// SIMATIC STEP 7 (V5.x) project S7_Mafra
// CPU: CPU 312
// CPU: CPU 312
// station: P_ADR_BUS
// station: Hardware
// station: Mafra_Praha
// station: P_ADR_BUS
// station: Hardware
// station: Mafra_Olomouc
// station: P_ADR_BUS
// station: Configuration
// station: P_ADR_BUS
// station: Configuration
// program: S7 Program(2)
// program: S7 Program(2)

SYMBOL_TABLE
"Události"	DB 100	DB 100
"DB_Chyby"	DB 101	DB 101
"DB_Ruèni povely pro HMI"	DB 120	DB 120
"DB_Data Hmi"	DB 140	DB 140
"Globální øízení"	FC 10	FC 10
"Váleèkové dopravníky"	FC 20	FC 20
"Data HMI"	FC 30	FC 30
"Chyby"	FC 40	FC 40
"Komunikace"	FC 50	FC 50
"Pohony P1,P2.1 a P2.2 OK"	I 0.0	BOOL	// Pohony dopr.P1 , toèny P2.2 a dopravníku P2.2 jsou OK
"Pohony P3,P4.1 a P4.2 OK"	I 0.1	BOOL	// Pohony dopr.P3 , toèny P4.1 a dopravníku P4.2 jsou OK
"Pohony P7,P8,P9 OK"	I 0.2	BOOL	// Pohony dopr.P7,P8,P9 jsou OK
"Silovka OK"	I 0.3	BOOL	// Silové obvody zapnuty
"Reset"	I 0.4	BOOL	// Reset programu
"Vynut NOT-Aus rozvadìè"	I 0.5	BOOL	// Vypnutý hlavní NOT-AUS na rozvadìèi
"NOT-AUS 1"	I 0.6	BOOL	// Vypnut NOT-AUS 1
"NOT-AUS 2"	I 0.7	BOOL	// Vypnut NOT-AUS 2
"Balík na konci P1"	I 1.0	BOOL	// Balík dojet na konci dopravníku 1
"Balík na konci P2.2"	I 1.1	BOOL	// Balík dojet na konci dopravníku 2.2
"Toèna 2.1 nájezd"	I 1.2	BOOL	// Toèna P2.1 pozice nájezd
"Toèna 2.1 výjezd"	I 1.3	BOOL	// Toèna P2.1 pozice výjezd
"Balík na konci P3"	I 1.4	BOOL	// Balík dojet na konci dopravníku 3
"Balík na konci P4.2"	I 1.5	BOOL	// Balík dojet na konci dopravníku 4.2
"Toèna 4.1 nájezd"	I 1.6	BOOL	// Toèna P4.1 pozice nájezd
"Toèna 4.1 výjezd"	I 1.7	BOOL	// Toèna P4.1 pozice výjezd
"Balík na konci P5"	I 2.0	BOOL	// Balík dojet na konci dopravníku 5
"Balík na konci P6"	I 2.1	BOOL	// Balík dojet na konci dopravníku 6
"Balík na konci P7"	I 2.2	BOOL	// Balík dojet na konci dopravníku 7
"Balík na konci P8"	I 2.3	BOOL	// Balík dojet na konci dopravníku 8
"S024"	I 2.4	BOOL	// stop na D2
"rezerva 1"	I 2.5	BOOL
"rezerva 2"	I 2.6	BOOL
"rezerva 3"	I 2.7	BOOL
"Komunikace vstup 1"	I 3.0	BOOL
"Komunikace vstup2"	I 3.1	BOOL
"Komunikace vstup 3"	I 3.2	BOOL
"Komunikace vstup 4"	I 3.3	BOOL
"rezerva 4"	I 3.4	BOOL
"rezerva 5"	I 3.5	BOOL
"rezerva 6"	I 3.6	BOOL
"rezerva 7"	I 3.7	BOOL
"True"	M 0.3	BOOL
"Automat"	M 1.0	BOOL	// Automatický chod stroje
"Chyba"	M 2.0	BOOL	// vyhlašení chybového stavu stroje
"PM21"	M 2.1	BOOL	// pomocný merkr
"Houkat"	M 4.4	BOOL	// pomocný merkr pro houkaèku
"Toèna P2 Stop nájezd"	M 6.0	BOOL
"Toèna P2 Stop výjezd"	M 6.1	BOOL
"Toèna P4 Stop nájezd"	M 6.2	BOOL
"Toèna P4 Stop výjezd"	M 6.4	BOOL
"M-Toèna 2 nájezd"	M 7.0	BOOL
"M-Toèna 2 výjezd"	M 7.1	BOOL
"M-Toèna 4 výjezd"	M 7.2	BOOL
"M-Toèna 4 nájezd"	M 7.3	BOOL
"Pøesun Balièka-P1"	M 20.0	BOOL	// pomocny merk pøesunu balíku z balièky na toènu
"Pøesun z Toèny na P3"	M 20.1	BOOL	// set a reset pøesunu balíku z toèny na dopravník P3
"Pøesun P3 - Toèna P4."	M 20.2	BOOL	// set a reset pøesunu z dopravníku P3 na toènu P4.1
"Pøesun Toèna P4.1-P5"	M 20.3	BOOL	// set a reset pøesunu z Toèny P4.1 na dopravník P5
"Pøesun P5-P6"	M 20.4	BOOL	// set a reset pøesunu balíku z P5 na P6
"Pøesun P6-P7"	M 20.5	BOOL	// set a reset pøesunu z dopravníku P6 na P7
"Pøesun P7-P8"	M 20.6	BOOL	// set a reset pøesunu z dopravníku P7 na P8
"CYC_INT5"	OB 35	OB 35	// Cyclic Interrupt 5
"I/O_FLT1"	OB 82	OB 82	// I/O Point Fault 1
"OBNL_FLT"	OB 85	OB 85	// OB Not Loaded Fault
"RACK_FLT"	OB 86	OB 86	// Loss of Rack Fault
"Complete Restart"	OB 100	OB 100
"Programming Error"	OB 121	OB 121
"Module Access Error"	OB 122	OB 122
"Dopravník 1 vpøed"	Q 4.0	BOOL	// Start dopravníku 1
"Toèna P2.1 nájezd"	Q 4.1	BOOL	// Toèna P2.1 nájezd
"Toèna P2.1 výjezd"	Q 4.2	BOOL	// Toèna P2.1 výjezd
"Toèna P2.1 brzda"	Q 4.3	BOOL	// Toèna P2.1 bzrda
"Dopravník 2.2 vpøed"	Q 4.4	BOOL	// Start dopravníku 2.2
"Dopravník 3 vpøed"	Q 4.5	BOOL	// Start dopravníku 3
"Toèna P4.1 nájezd"	Q 4.6	BOOL	// Toèna P4.1 nájezd
"Toèna P4.1 výjezd"	Q 4.7	BOOL	// Toèna P4.1 výjezd
"Toèna P4.1 brzda"	Q 5.0	BOOL	// Toèna P4.1 bzrda
"Dopravník P4.2 vpøed"	Q 5.1	BOOL	// Start dopravníku 4.2
"Dopravník 5 vpøed"	Q 5.2	BOOL	// Start dopravníku 5
"Dopravník 6 vpøed"	Q 5.3	BOOL	// Start dopravníku 6
"Dopravník 7 vpøed"	Q 5.4	BOOL	// Start dopravníku 7
"Dopravník 8 vpøed"	Q 5.5	BOOL	// Start dopravníku 8
"rezerva 8"	Q 5.6	BOOL
"rezerva 9"	Q 5.7	BOOL
"Signálka Zapnuto"	Q 6.0	BOOL	// Signálk zapnuto
"rezerva 10"	Q 6.1	BOOL
"rezerva 11"	Q 6.2	BOOL
"rezerva 12"	Q 6.3	BOOL
"Maják zelená"	Q 6.4	BOOL	// Signalizaèní sloupek - zelená
"Maják oranžová"	Q 6.5	BOOL	// Signalizaèní sloupek - oranžová
"Maják èervená"	Q 6.6	BOOL	// Signalizaèní sloupek - èervená
"Houkaèka"	Q 6.7	BOOL	// Signalizaèní sloupek - houkaèka
"Komunikace výstup 1"	Q 7.0	BOOL
"Komunikace výstup 2"	Q 7.1	BOOL
"Komunikace výstup 3"	Q 7.2	BOOL
"Komunikace-Plná linka"	Q 7.3	BOOL
"rezerva 13"	Q 7.4	BOOL
"rezerva 14"	Q 7.5	BOOL
"rezerva 15"	Q 7.6	BOOL
"rezerva 16"	Q 7.7	BOOL
"T-Automat"	T 0	TIMER	// zpoždìné spuštìní automatu
"T-Balík na konci P8"	T 2	TIMER	// Zpoždìný start pøesunu
"T-Pozor"	T 3	TIMER	// upozornìní na spouštìjící se automat
"T-S011"	T 10	TIMER	// balik dojet na konci D2
"T-S015"	T 11	TIMER
"T-Balík na konci"	T 12	TIMER
"T-Možno otoèit toènu"	T 13	TIMER
"T-Možno otoèit toènu P4"	T 14	TIMER
"T-S010"	T 15	TIMER	// balík dojet na konci skluzu
"T-Pøesun Balièka-P2.2"	T 20	TIMER	// èasovaè pro vyhlášení pøíliš dlouhého pøesunu
"T-Pøesun P2.2-P3"	T 21	TIMER	// èasovaè pro vyhlášení pøíliš dlouhého pøesunu
"T-Pøesun P3-P4.2"	T 22	TIMER	// èasovaè pro vyhlášení pøíliš dlouhého pøesunu
"T-Pøesun P4.2-P5"	T 23	TIMER	// èasovaè pro vyhlášení pøíliš dlouhého pøesunu
"T-Pøesun P5-P6"	T 24	TIMER	// èasovaè pro vyhlášení pøíliš dlouhého pøesunu
"T-Pøesun P6-P7"	T 25	TIMER	// èasovaè pro vyhlášení pøíliš dlouhého pøesunu
"T-Pøesun P7-P8"	T 26	TIMER	// èasovaè pro vyhlášení pøíliš dlouhého pøesunu
"T-Otaèení Toèny P2.1"	T 27	TIMER	// èasovaè pro vyhlášení pøíliš dlouhého otáèení toèny
"T-Otáèení toèny P4.1"	T 28	TIMER	// èasovaè pro vyhlášení pøíliš dlouhého otáèení toèny
"T-S014"	T 30	TIMER	// balik dojet na konci dopravniku
"T--S015"	T 31	TIMER	// balík na konci D4
"T-S020"	T 32	TIMER	// balík na konci D5
"T-S021"	T 33	TIMER	// balík na konci D6
"T-S022"	T 34	TIMER	// balík na konci D7
"T--S011"	T 35	TIMER
"T-S024"	T 37	TIMER	// Stop na D2
"VAT_1"	VAT 1	
END_SYMBOL_TABLE

FUNCTION "Globální øízení" : VOID	// FC 10
VERSION : 0.1
BEGIN
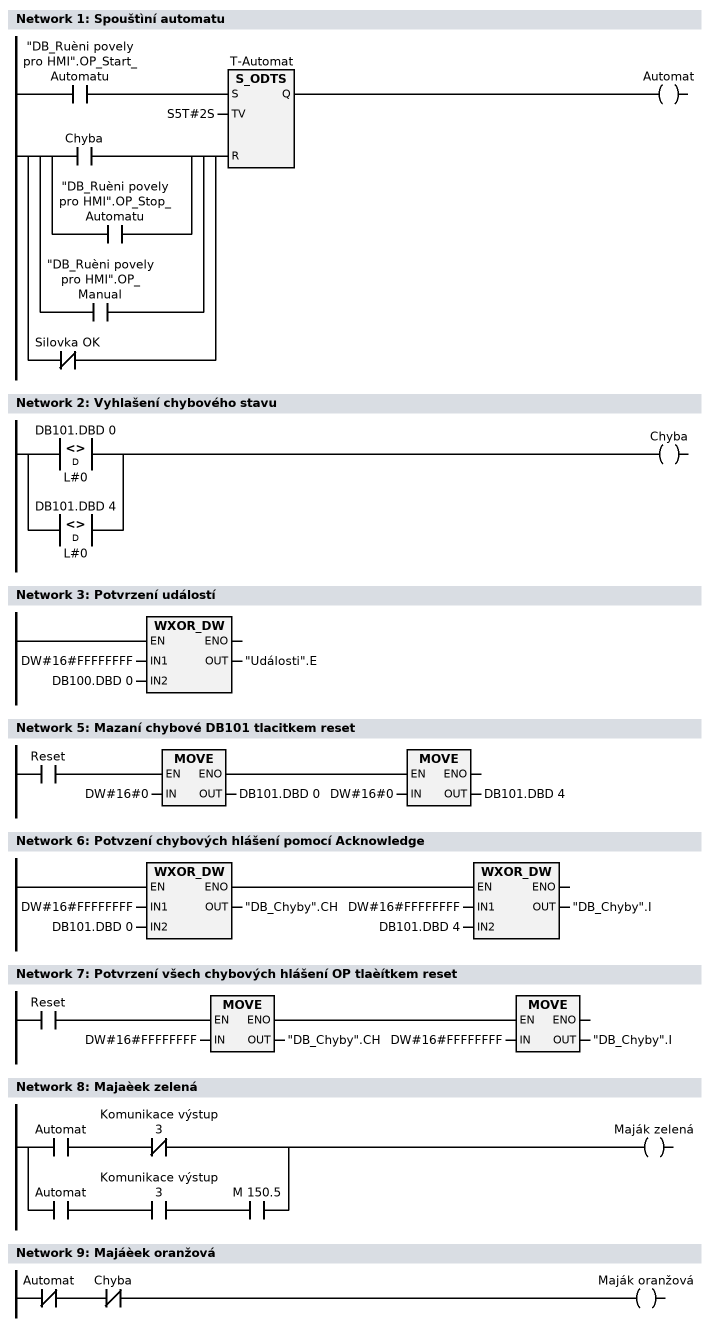
NETWORK
TITLE = Spouštìní automatu 
      A     "DB_Ruèni povely pro HMI".OP_Start_Automatu;
      L     S5T#2S;
      SS    "T-Automat";
      A(;
      O     "Chyba";
      O     "DB_Ruèni povely pro HMI".OP_Stop_Automatu;
      O     "DB_Ruèni povely pro HMI".OP_Manual;
      ON    "Silovka OK";
      );
      R     "T-Automat";
      NOP   0;
      NOP   0;
      A     "T-Automat";
      =     "Automat";
NETWORK
TITLE = Vyhlašení chybového stavu 
      O(;
      L     DB101.DBD 0;
      L     L#0;
      <>D;
      );
      O(;
      L     DB101.DBD 4;
      L     L#0;
      <>D;
      );
      =     "Chyba";
NETWORK
TITLE = Potvrzení událostí
      L     DW#16#FFFFFFFF;
      L     DB100.DBD 0;
      XOD;
      T     "Události".E;
      NOP   0;
NETWORK
TITLE = Akustická signalizace 
      A(;
      O(;
      A     "Chyba";
      FP    "PM21";
      S     "Houkat";
      A     "Reset";
      R     "Houkat";
      A     "Houkat";
      );
      O(;
      A     "DB_Ruèni povely pro HMI".OP_Start_Automatu;
      L     S5T#2S;
      SE    "T-Pozor";
      A(;
      O     "Chyba";
      O     "DB_Ruèni povely pro HMI".OP_Manual;
      O     "DB_Ruèni povely pro HMI".OP_Stop_Automatu;
      O     "Automat";
      );
      R     "T-Pozor";
      NOP   0;
      NOP   0;
      A     "T-Pozor";
      );
      );
      A     M 150.5;
      =     "Houkaèka";
NETWORK
TITLE = Mazaní chybové DB101 tlacitkem reset
      A(;
      A     "Reset";
      JNB   _001;
      L     DW#16#0;
      T     DB101.DBD 0;
      SET;
      SAVE;
      CLR;
_001: A     BR;
      );
      JNB   _002;
      L     DW#16#0;
      T     DB101.DBD 4;
_002: NOP   0;
NETWORK
TITLE = Potvzení chybových hlášení pomocí Acknowledge
      A(;
      L     DW#16#FFFFFFFF;
      L     DB101.DBD 0;
      XOD;
      T     "DB_Chyby".CH;
      SET;
      SAVE;
      CLR;
      A     BR;
      );
      JNB   _003;
      L     DW#16#FFFFFFFF;
      L     DB101.DBD 4;
      XOD;
      T     "DB_Chyby".I;
_003: NOP   0;
NETWORK
TITLE = Potvrzení všech chybových hlášení OP tlaèítkem reset
      A(;
      A     "Reset";
      JNB   _004;
      L     DW#16#FFFFFFFF;
      T     "DB_Chyby".CH;
      SET;
      SAVE;
      CLR;
_004: A     BR;
      );
      JNB   _005;
      L     DW#16#FFFFFFFF;
      T     "DB_Chyby".I;
_005: NOP   0;
NETWORK
TITLE = Majaèek zelená 
      A     "Automat";
      AN    "Komunikace výstup 3";
      O;
      A     "Automat";
      A     "Komunikace výstup 3";
      A     M 150.5;
      =     "Maják zelená";
NETWORK
TITLE = Majáèek oranžová 
      AN    "Automat";
      AN    "Chyba";
      =     "Maják oranžová";
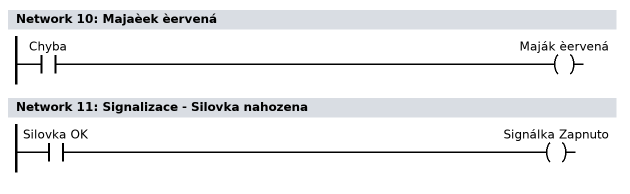
NETWORK
TITLE = Majaèek èervená 
      A     "Chyba";
      =     "Maják èervená";
NETWORK
TITLE = Signalizace - Silovka nahozena
      A     "Silovka OK";
      =     "Signálka Zapnuto";
END_FUNCTION

FUNCTION "Váleèkové dopravníky" : VOID	// FC 20
VERSION : 0.1
BEGIN
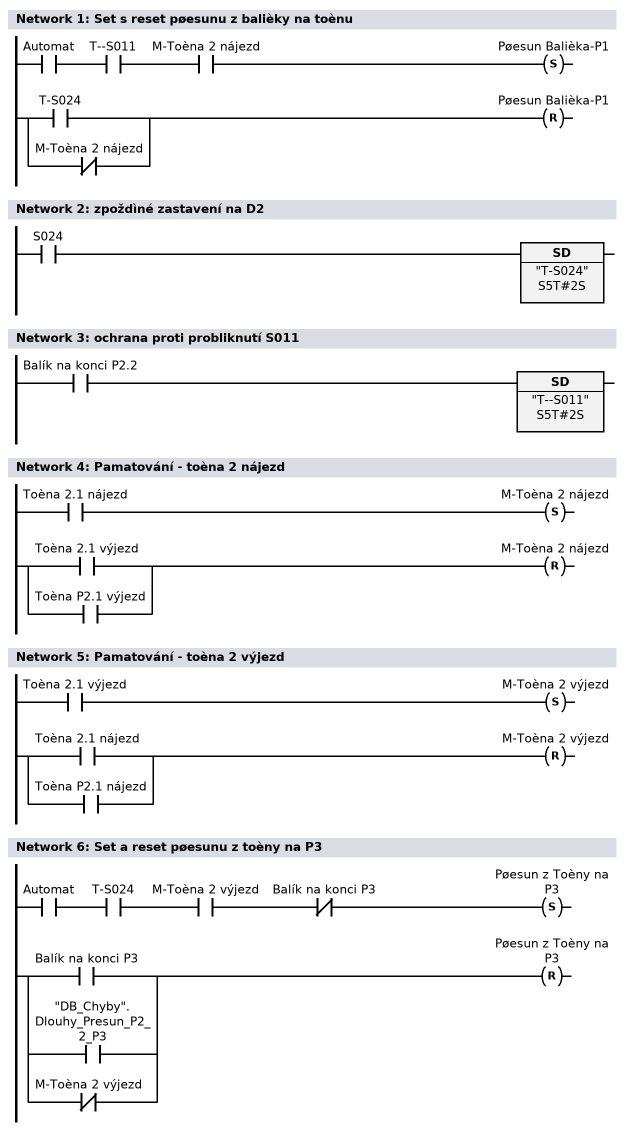
NETWORK
TITLE = Set s reset pøesunu z balièky na toènu
      A     "Automat";
      A     "T--S011";
      A     "M-Toèna 2 nájezd";
      S     "Pøesun Balièka-P1";
      A(;
      O     "T-S024";
      ON    "M-Toèna 2 nájezd";
      );
      R     "Pøesun Balièka-P1";
      NOP   0;
NETWORK
TITLE = zpoždìné zastavení na D2
      A     "S024";
      L     S5T#2S;
      SD    "T-S024";
NETWORK
TITLE = ochrana proti probliknutí S011
      A     "Balík na konci P2.2";
      L     S5T#2S;
      SD    "T--S011";
NETWORK
TITLE = Pamatování - toèna 2 nájezd
      A     "Toèna 2.1 nájezd";
      S     "M-Toèna 2 nájezd";
      A(;
      O     "Toèna 2.1 výjezd";
      O     "Toèna P2.1 výjezd";
      );
      R     "M-Toèna 2 nájezd";
      NOP   0;
NETWORK
TITLE = Pamatování - toèna 2 výjezd
      A     "Toèna 2.1 výjezd";
      S     "M-Toèna 2 výjezd";
      A(;
      O     "Toèna 2.1 nájezd";
      O     "Toèna P2.1 nájezd";
      );
      R     "M-Toèna 2 výjezd";
      NOP   0;
NETWORK
TITLE = Set a reset pøesunu z toèny na P3
      A     "Automat";
      A     "T-S024";
      A     "M-Toèna 2 výjezd";
      AN    "Balík na konci P3";
      S     "Pøesun z Toèny na P3";
      A(;
      O     "Balík na konci P3";
      O     "DB_Chyby".Dlouhy_Presun_P2_2_P3;
      ON    "M-Toèna 2 výjezd";
      );
      R     "Pøesun z Toèny na P3";
      NOP   0;
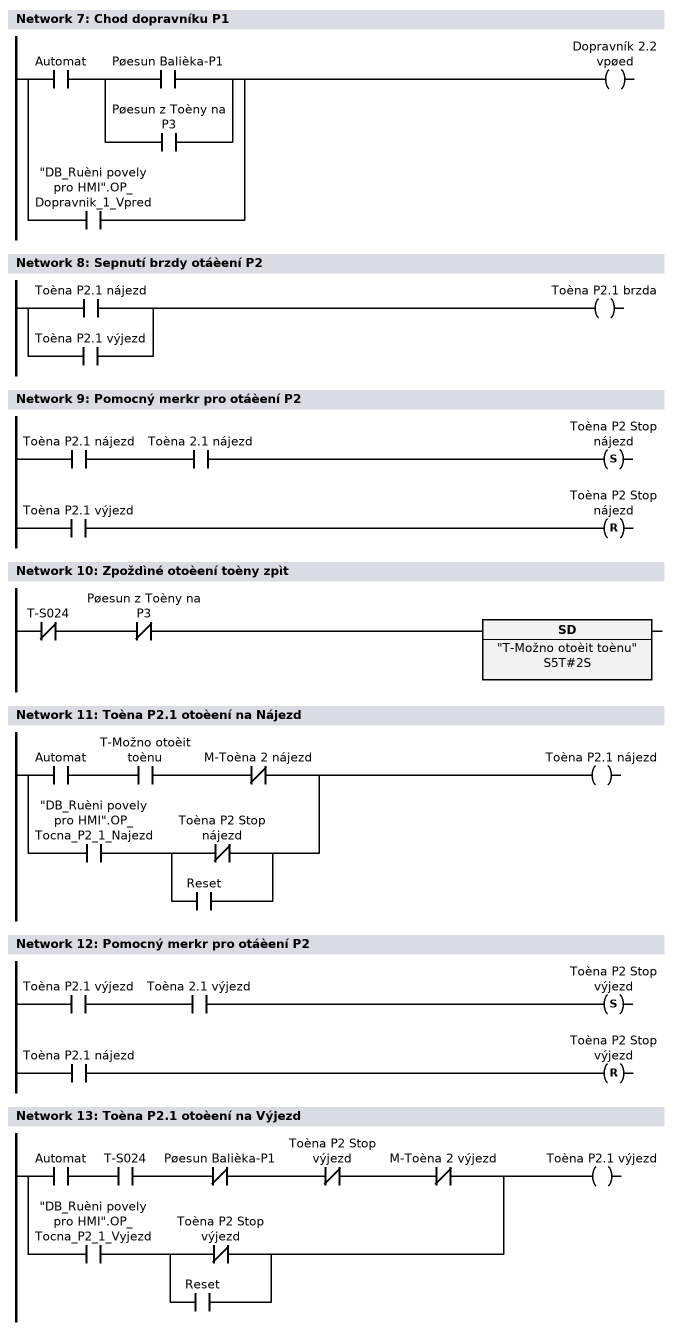
NETWORK
TITLE = Chod dopravníku P1
      A     "Automat";
      A(;
      O     "Pøesun Balièka-P1";
      O     "Pøesun z Toèny na P3";
      );
      O     "DB_Ruèni povely pro HMI".OP_Dopravnik_1_Vpred;
      =     "Dopravník 2.2 vpøed";
NETWORK
TITLE = Sepnutí brzdy otáèení P2
      O     "Toèna P2.1 nájezd";
      O     "Toèna P2.1 výjezd";
      =     "Toèna P2.1 brzda";
NETWORK
TITLE = Pomocný merkr pro otáèení P2
//Kvùli prokmitu toèny 
      A     "Toèna P2.1 nájezd";
      A     "Toèna 2.1 nájezd";
      S     "Toèna P2 Stop nájezd";
      A     "Toèna P2.1 výjezd";
      R     "Toèna P2 Stop nájezd";
      NOP   0;
NETWORK
TITLE = Zpoždìné otoèení toèny zpìt
      AN    "T-S024";
      AN    "Pøesun z Toèny na P3";
      L     S5T#2S;
      SD    "T-Možno otoèit toènu";
NETWORK
TITLE = Toèna P2.1 otoèení na Nájezd
      A     "Automat";
      A     "T-Možno otoèit toènu";
      AN    "M-Toèna 2 nájezd";
      O;
      A     "DB_Ruèni povely pro HMI".OP_Tocna_P2_1_Najezd;
      A(;
      ON    "Toèna P2 Stop nájezd";
      O     "Reset";
      );
      =     "Toèna P2.1 nájezd";
NETWORK
TITLE = Pomocný merkr pro otáèení P2
//Kvùli prokmitu toèny 
      A     "Toèna P2.1 výjezd";
      A     "Toèna 2.1 výjezd";
      S     "Toèna P2 Stop výjezd";
      A     "Toèna P2.1 nájezd";
      R     "Toèna P2 Stop výjezd";
      NOP   0;
NETWORK
TITLE = Toèna P2.1 otoèení na Výjezd
      A     "Automat";
      A     "T-S024";
      AN    "Pøesun Balièka-P1";
      AN    "Toèna P2 Stop výjezd";
      AN    "M-Toèna 2 výjezd";
      O;
      A     "DB_Ruèni povely pro HMI".OP_Tocna_P2_1_Vyjezd;
      A(;
      ON    "Toèna P2 Stop výjezd";
      O     "Reset";
      );
      =     "Toèna P2.1 výjezd";
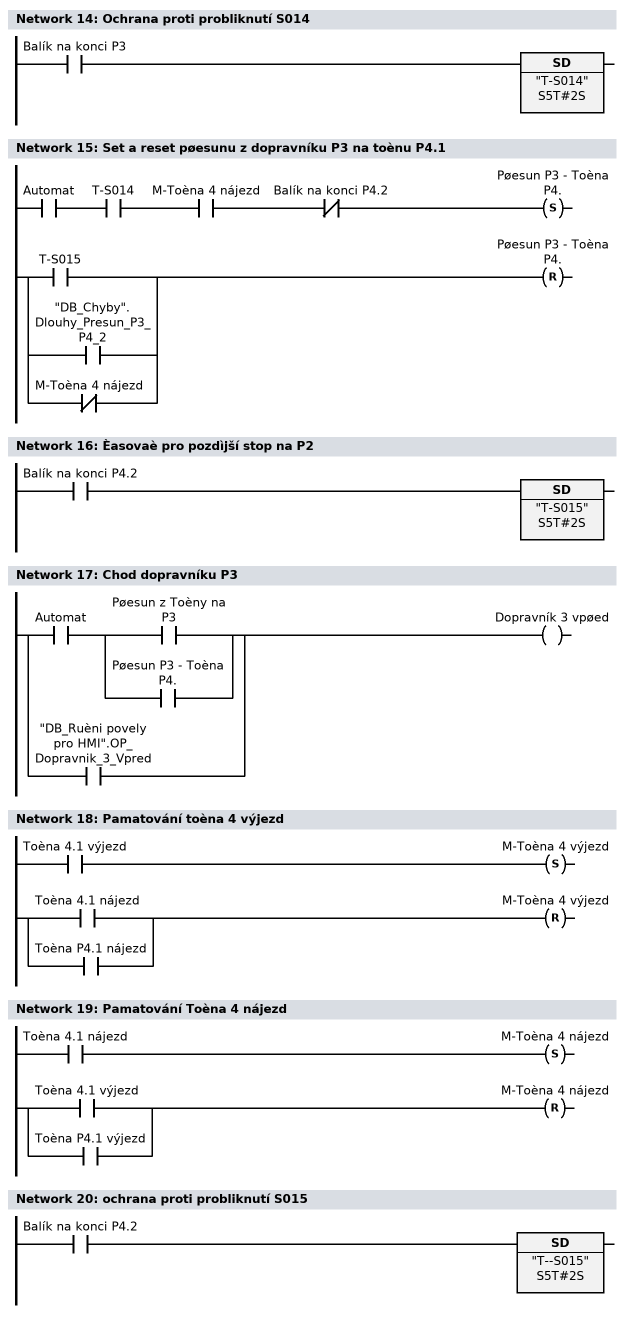
NETWORK
TITLE = Ochrana proti probliknutí S014
      A     "Balík na konci P3";
      L     S5T#2S;
      SD    "T-S014";
NETWORK
TITLE = Set a reset pøesunu z dopravníku P3 na toènu P4.1
      A     "Automat";
      A     "T-S014";
      A     "M-Toèna 4 nájezd";
      AN    "Balík na konci P4.2";
      S     "Pøesun P3 - Toèna P4.";
      A(;
      O     "T-S015";
      O     "DB_Chyby".Dlouhy_Presun_P3_P4_2;
      ON    "M-Toèna 4 nájezd";
      );
      R     "Pøesun P3 - Toèna P4.";
      NOP   0;
NETWORK
TITLE = Èasovaè pro pozdìjší stop na P2
      A     "Balík na konci P4.2";
      L     S5T#2S;
      SD    "T-S015";
NETWORK
TITLE = Chod dopravníku P3
      A     "Automat";
      A(;
      O     "Pøesun z Toèny na P3";
      O     "Pøesun P3 - Toèna P4.";
      );
      O     "DB_Ruèni povely pro HMI".OP_Dopravnik_3_Vpred;
      =     "Dopravník 3 vpøed";
NETWORK
TITLE = Pamatování toèna 4 výjezd
      A     "Toèna 4.1 výjezd";
      S     "M-Toèna 4 výjezd";
      A(;
      O     "Toèna 4.1 nájezd";
      O     "Toèna P4.1 nájezd";
      );
      R     "M-Toèna 4 výjezd";
      NOP   0;
NETWORK
TITLE = Pamatování Toèna 4 nájezd
      A     "Toèna 4.1 nájezd";
      S     "M-Toèna 4 nájezd";
      A(;
      O     "Toèna 4.1 výjezd";
      O     "Toèna P4.1 výjezd";
      );
      R     "M-Toèna 4 nájezd";
      NOP   0;
NETWORK
TITLE = ochrana proti probliknutí S015
      A     "Balík na konci P4.2";
      L     S5T#2S;
      SD    "T--S015";
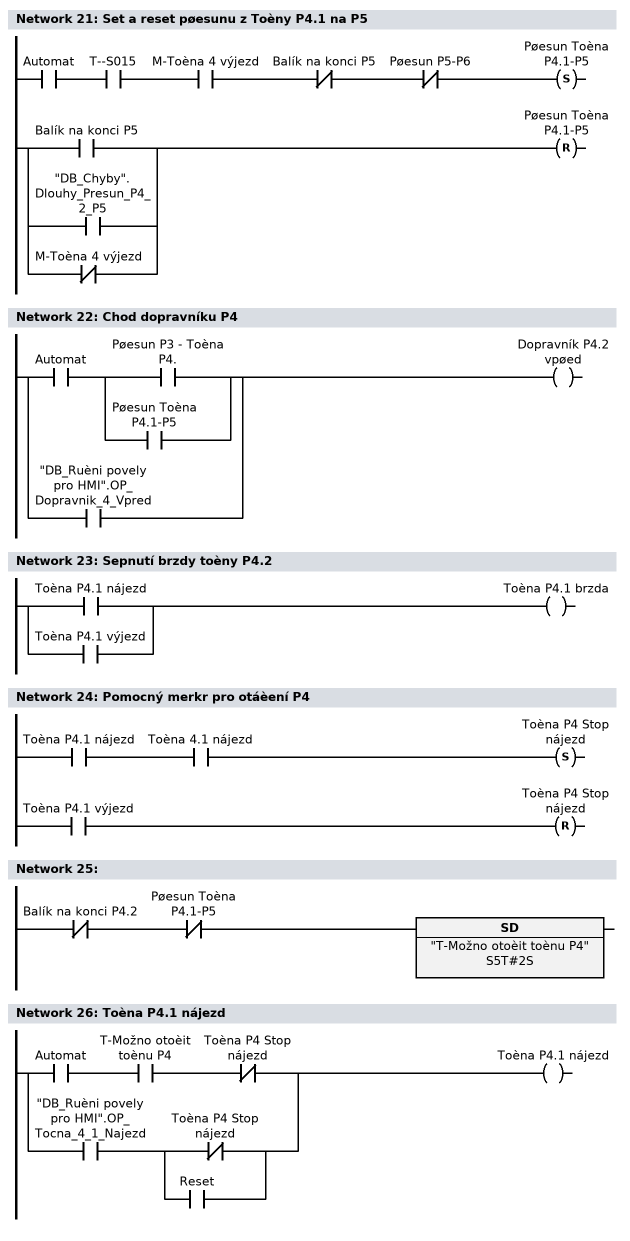
NETWORK
TITLE = Set a reset pøesunu z Toèny P4.1 na P5
      A     "Automat";
      A     "T--S015";
      A     "M-Toèna 4 výjezd";
      AN    "Balík na konci P5";
      AN    "Pøesun P5-P6";
      S     "Pøesun Toèna P4.1-P5";
      A(;
      O     "Balík na konci P5";
      O     "DB_Chyby".Dlouhy_Presun_P4_2_P5;
      ON    "M-Toèna 4 výjezd";
      );
      R     "Pøesun Toèna P4.1-P5";
      NOP   0;
NETWORK
TITLE = Chod dopravníku P4
      A     "Automat";
      A(;
      O     "Pøesun P3 - Toèna P4.";
      O     "Pøesun Toèna P4.1-P5";
      );
      O     "DB_Ruèni povely pro HMI".OP_Dopravnik_4_Vpred;
      =     "Dopravník P4.2 vpøed";
NETWORK
TITLE = Sepnutí brzdy toèny P4.2
      O     "Toèna P4.1 nájezd";
      O     "Toèna P4.1 výjezd";
      =     "Toèna P4.1 brzda";
NETWORK
TITLE = Pomocný merkr pro otáèení P4
//
//Kvùli prokmitu toèny 
      A     "Toèna P4.1 nájezd";
      A     "Toèna 4.1 nájezd";
      S     "Toèna P4 Stop nájezd";
      A     "Toèna P4.1 výjezd";
      R     "Toèna P4 Stop nájezd";
      NOP   0;
NETWORK
TITLE =
      AN    "Balík na konci P4.2";
      AN    "Pøesun Toèna P4.1-P5";
      L     S5T#2S;
      SD    "T-Možno otoèit toènu P4";
NETWORK
TITLE = Toèna P4.1 nájezd
      A     "Automat";
      A     "T-Možno otoèit toènu P4";
      AN    "Toèna P4 Stop nájezd";
      O;
      A     "DB_Ruèni povely pro HMI".OP_Tocna_4_1_Najezd;
      A(;
      ON    "Toèna P4 Stop nájezd";
      O     "Reset";
      );
      =     "Toèna P4.1 nájezd";
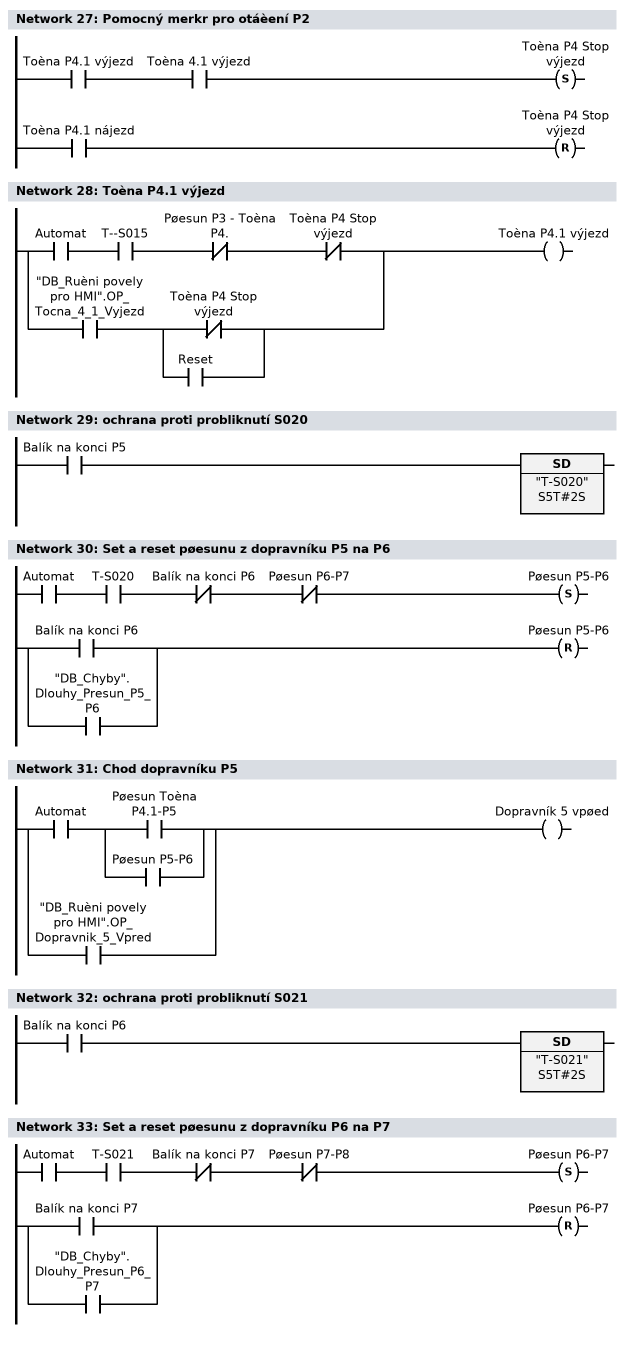
NETWORK
TITLE = Pomocný merkr pro otáèení P2
//Kvùli prokmitu toèny 
      A     "Toèna P4.1 výjezd";
      A     "Toèna 4.1 výjezd";
      S     "Toèna P4 Stop výjezd";
      A     "Toèna P4.1 nájezd";
      R     "Toèna P4 Stop výjezd";
      NOP   0;
NETWORK
TITLE = Toèna P4.1 výjezd
      A     "Automat";
      A     "T--S015";
      AN    "Pøesun P3 - Toèna P4.";
      AN    "Toèna P4 Stop výjezd";
      O;
      A     "DB_Ruèni povely pro HMI".OP_Tocna_4_1_Vyjezd;
      A(;
      ON    "Toèna P4 Stop výjezd";
      O     "Reset";
      );
      =     "Toèna P4.1 výjezd";
NETWORK
TITLE = ochrana proti probliknutí S020
      A     "Balík na konci P5";
      L     S5T#2S;
      SD    "T-S020";
NETWORK
TITLE = Set a reset pøesunu z dopravníku P5 na P6
      A     "Automat";
      A     "T-S020";
      AN    "Balík na konci P6";
      AN    "Pøesun P6-P7";
      S     "Pøesun P5-P6";
      A(;
      O     "Balík na konci P6";
      O     "DB_Chyby".Dlouhy_Presun_P5_P6;
      );
      R     "Pøesun P5-P6";
      NOP   0;
NETWORK
TITLE = Chod dopravníku P5
      A     "Automat";
      A(;
      O     "Pøesun Toèna P4.1-P5";
      O     "Pøesun P5-P6";
      );
      O     "DB_Ruèni povely pro HMI".OP_Dopravnik_5_Vpred;
      =     "Dopravník 5 vpøed";
NETWORK
TITLE = ochrana proti probliknutí S021
      A     "Balík na konci P6";
      L     S5T#2S;
      SD    "T-S021";
NETWORK
TITLE = Set a reset pøesunu z dopravníku P6 na P7
      A     "Automat";
      A     "T-S021";
      AN    "Balík na konci P7";
      AN    "Pøesun P7-P8";
      S     "Pøesun P6-P7";
      A(;
      O     "Balík na konci P7";
      O     "DB_Chyby".Dlouhy_Presun_P6_P7;
      );
      R     "Pøesun P6-P7";
      NOP   0;
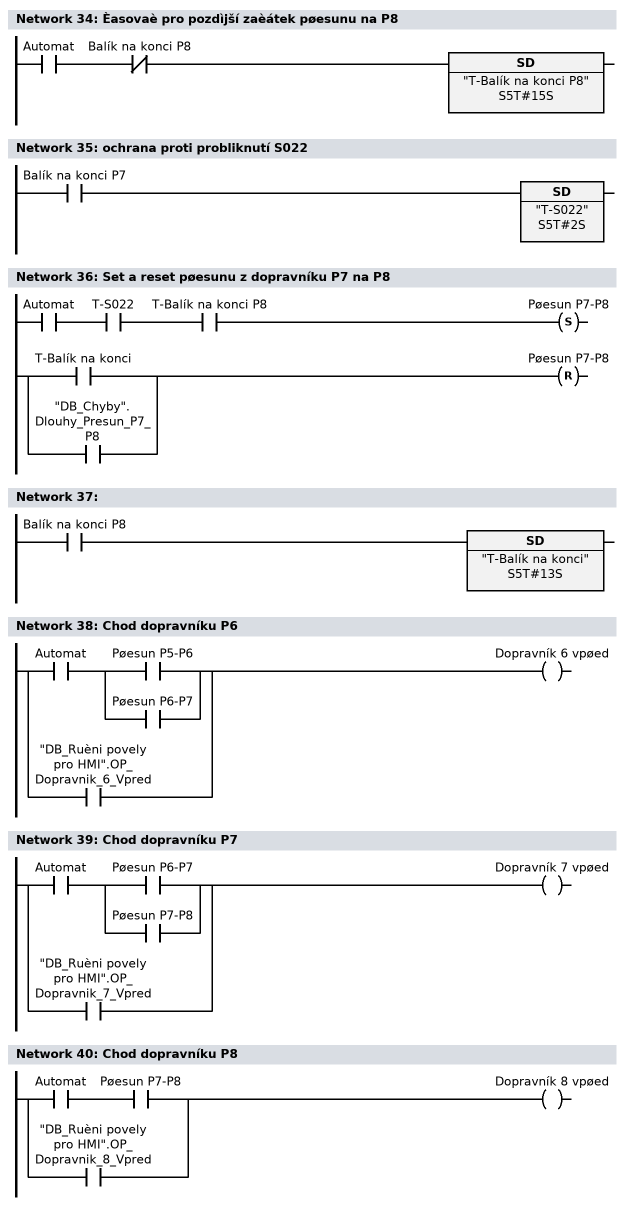
NETWORK
TITLE = Èasovaè pro pozdìjší zaèátek pøesunu na P8
//Je to z dùvodu dání èasu obsluze vozíku na odebrání pøedchozího balíku
      A     "Automat";
      AN    "Balík na konci P8";
      L     S5T#15S;
      SD    "T-Balík na konci P8";
NETWORK
TITLE = ochrana proti probliknutí S022
      A     "Balík na konci P7";
      L     S5T#2S;
      SD    "T-S022";
NETWORK
TITLE = Set a reset pøesunu z dopravníku P7 na P8
      A     "Automat";
      A     "T-S022";
      A     "T-Balík na konci P8";
      S     "Pøesun P7-P8";
      A(;
      O     "T-Balík na konci";
      O     "DB_Chyby".Dlouhy_Presun_P7_P8;
      );
      R     "Pøesun P7-P8";
      NOP   0;
NETWORK
TITLE =
      A     "Balík na konci P8";
      L     S5T#13S;
      SD    "T-Balík na konci";
NETWORK
TITLE = Chod dopravníku P6
      A     "Automat";
      A(;
      O     "Pøesun P5-P6";
      O     "Pøesun P6-P7";
      );
      O     "DB_Ruèni povely pro HMI".OP_Dopravnik_6_Vpred;
      =     "Dopravník 6 vpøed";
NETWORK
TITLE = Chod dopravníku P7
      A     "Automat";
      A(;
      O     "Pøesun P6-P7";
      O     "Pøesun P7-P8";
      );
      O     "DB_Ruèni povely pro HMI".OP_Dopravnik_7_Vpred;
      =     "Dopravník 7 vpøed";
NETWORK
TITLE = Chod dopravníku P8
      A     "Automat";
      A     "Pøesun P7-P8";
      O     "DB_Ruèni povely pro HMI".OP_Dopravnik_8_Vpred;
      =     "Dopravník 8 vpøed";
END_FUNCTION

FUNCTION "Data HMI" : VOID	// FC 30
VERSION : 0.1
BEGIN
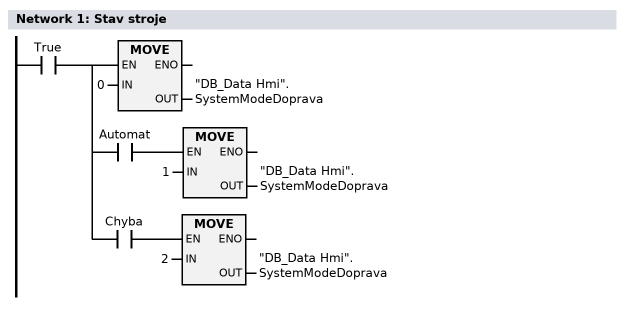
NETWORK
TITLE = Stav stroje 
      A     "True";
      =     L 0.0;
      A     L 0.0;
      JNB   _001;
      L     0;
      T     "DB_Data Hmi".SystemModeDoprava;
_001: NOP   0;
      A     L 0.0;
      A     "Automat";
      JNB   _002;
      L     1;
      T     "DB_Data Hmi".SystemModeDoprava;
_002: NOP   0;
      A     L 0.0;
      A     "Chyba";
      JNB   _003;
      L     2;
      T     "DB_Data Hmi".SystemModeDoprava;
_003: NOP   0;
END_FUNCTION

FUNCTION "Chyby" : VOID	// FC 40
VERSION : 0.1
BEGIN
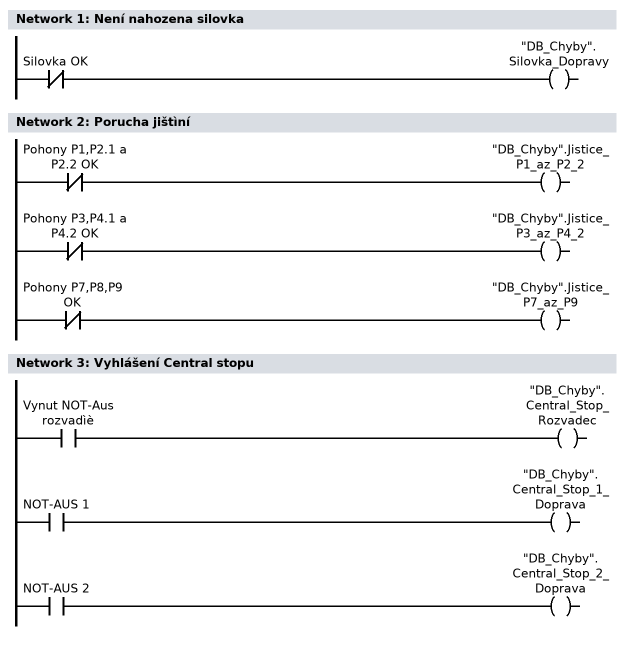
NETWORK
TITLE = Není nahozena silovka 
      AN    "Silovka OK";
      =     "DB_Chyby".Silovka_Dopravy;
NETWORK
TITLE = Porucha jištìní
      AN    "Pohony P1,P2.1 a P2.2 OK";
      =     "DB_Chyby".Jistice_P1_az_P2_2;
      AN    "Pohony P3,P4.1 a P4.2 OK";
      =     "DB_Chyby".Jistice_P3_az_P4_2;
      AN    "Pohony P7,P8,P9 OK";
      =     "DB_Chyby".Jistice_P7_az_P9;
NETWORK
TITLE = Vyhlášení Central stopu
      A     "Vynut NOT-Aus rozvadìè";
      =     "DB_Chyby".Central_Stop_Rozvadec;
      A     "NOT-AUS 1";
      =     "DB_Chyby".Central_Stop_1_Doprava;
      A     "NOT-AUS 2";
      =     "DB_Chyby".Central_Stop_2_Doprava;
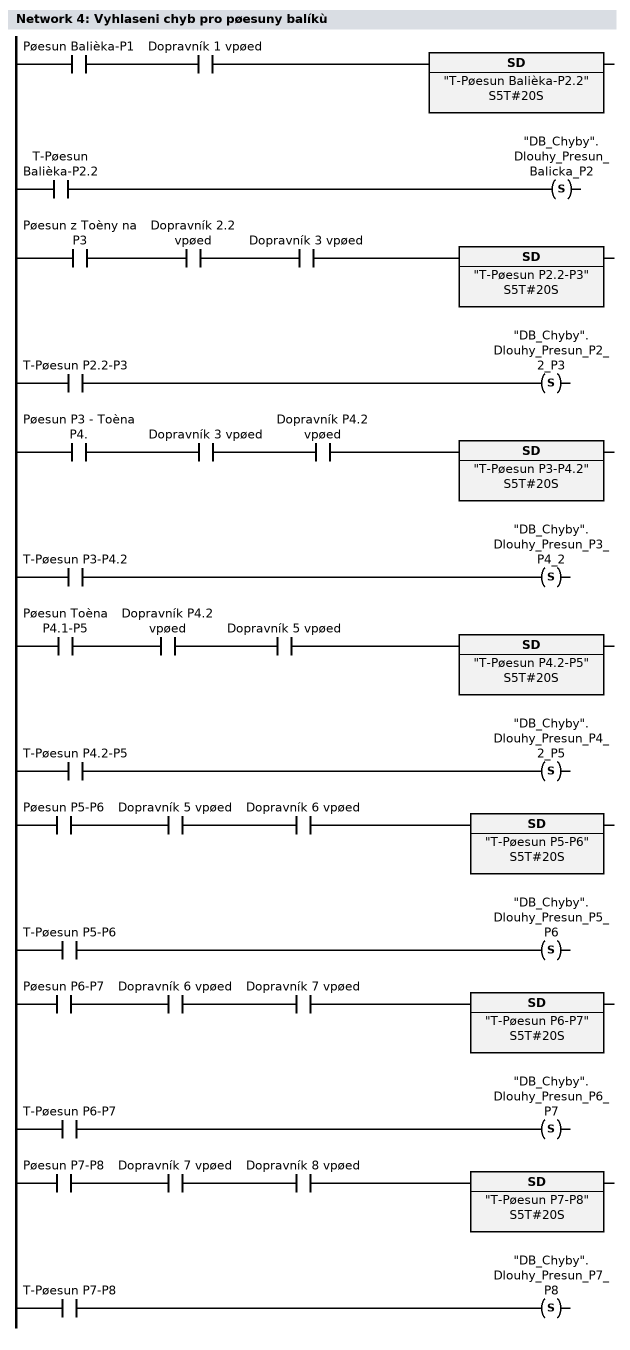
NETWORK
TITLE = Vyhlaseni chyb pro pøesuny balíkù
      A     "Pøesun Balièka-P1";
      A     "Dopravník 1 vpøed";
      L     S5T#20S;
      SD    "T-Pøesun Balièka-P2.2";
      A     "T-Pøesun Balièka-P2.2";
      S     "DB_Chyby".Dlouhy_Presun_Balicka_P2;
      A     "Pøesun z Toèny na P3";
      A     "Dopravník 2.2 vpøed";
      A     "Dopravník 3 vpøed";
      L     S5T#20S;
      SD    "T-Pøesun P2.2-P3";
      A     "T-Pøesun P2.2-P3";
      S     "DB_Chyby".Dlouhy_Presun_P2_2_P3;
      A     "Pøesun P3 - Toèna P4.";
      A     "Dopravník 3 vpøed";
      A     "Dopravník P4.2 vpøed";
      L     S5T#20S;
      SD    "T-Pøesun P3-P4.2";
      A     "T-Pøesun P3-P4.2";
      S     "DB_Chyby".Dlouhy_Presun_P3_P4_2;
      A     "Pøesun Toèna P4.1-P5";
      A     "Dopravník P4.2 vpøed";
      A     "Dopravník 5 vpøed";
      L     S5T#20S;
      SD    "T-Pøesun P4.2-P5";
      A     "T-Pøesun P4.2-P5";
      S     "DB_Chyby".Dlouhy_Presun_P4_2_P5;
      A     "Pøesun P5-P6";
      A     "Dopravník 5 vpøed";
      A     "Dopravník 6 vpøed";
      L     S5T#20S;
      SD    "T-Pøesun P5-P6";
      A     "T-Pøesun P5-P6";
      S     "DB_Chyby".Dlouhy_Presun_P5_P6;
      A     "Pøesun P6-P7";
      A     "Dopravník 6 vpøed";
      A     "Dopravník 7 vpøed";
      L     S5T#20S;
      SD    "T-Pøesun P6-P7";
      A     "T-Pøesun P6-P7";
      S     "DB_Chyby".Dlouhy_Presun_P6_P7;
      A     "Pøesun P7-P8";
      A     "Dopravník 7 vpøed";
      A     "Dopravník 8 vpøed";
      L     S5T#20S;
      SD    "T-Pøesun P7-P8";
      A     "T-Pøesun P7-P8";
      S     "DB_Chyby".Dlouhy_Presun_P7_P8;
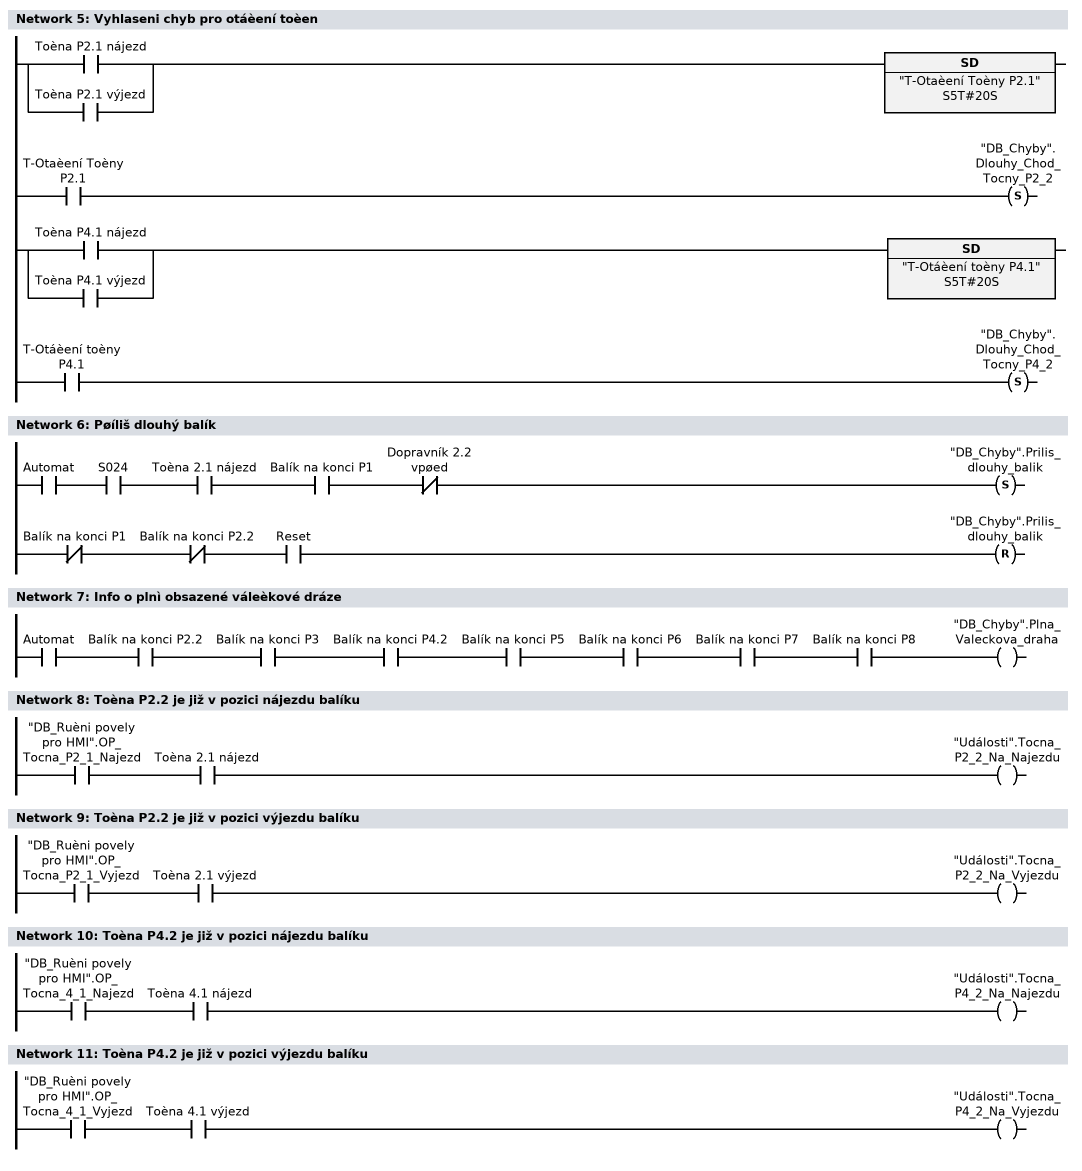
NETWORK
TITLE = Vyhlaseni chyb pro otáèení toèen
      A     "Toèna P2.1 nájezd";
      O;
      A     "Toèna P2.1 výjezd";
      L     S5T#20S;
      SD    "T-Otaèení Toèny P2.1";
      A     "T-Otaèení Toèny P2.1";
      S     "DB_Chyby".Dlouhy_Chod_Tocny_P2_2;
      A     "Toèna P4.1 nájezd";
      O;
      A     "Toèna P4.1 výjezd";
      L     S5T#20S;
      SD    "T-Otáèení toèny P4.1";
      A     "T-Otáèení toèny P4.1";
      S     "DB_Chyby".Dlouhy_Chod_Tocny_P4_2;
NETWORK
TITLE = Pøíliš dlouhý balík
//S010- má obrácenou logiku
      A     "Automat";
      A     "S024";
      A     "Toèna 2.1 nájezd";
      A     "Balík na konci P1";
      AN    "Dopravník 2.2 vpøed";
      S     "DB_Chyby".Prilis_dlouhy_balik;
      AN    "Balík na konci P1";
      AN    "Balík na konci P2.2";
      A     "Reset";
      R     "DB_Chyby".Prilis_dlouhy_balik;
      NOP   0;
NETWORK
TITLE = Info o plnì obsazené váleèkové dráze
      A     "Automat";
      A     "Balík na konci P2.2";
      A     "Balík na konci P3";
      A     "Balík na konci P4.2";
      A     "Balík na konci P5";
      A     "Balík na konci P6";
      A     "Balík na konci P7";
      A     "Balík na konci P8";
      =     "DB_Chyby".Plna_Valeckova_draha;
NETWORK
TITLE = Toèna P2.2 je již v pozici nájezdu balíku
      A     "DB_Ruèni povely pro HMI".OP_Tocna_P2_1_Najezd;
      A     "Toèna 2.1 nájezd";
      =     "Události".Tocna_P2_2_Na_Najezdu;
NETWORK
TITLE = Toèna P2.2 je již v pozici výjezdu balíku
      A     "DB_Ruèni povely pro HMI".OP_Tocna_P2_1_Vyjezd;
      A     "Toèna 2.1 výjezd";
      =     "Události".Tocna_P2_2_Na_Vyjezdu;
NETWORK
TITLE = Toèna P4.2 je již v pozici nájezdu balíku
      A     "DB_Ruèni povely pro HMI".OP_Tocna_4_1_Najezd;
      A     "Toèna 4.1 nájezd";
      =     "Události".Tocna_P4_2_Na_Najezdu;
NETWORK
TITLE = Toèna P4.2 je již v pozici výjezdu balíku
      A     "DB_Ruèni povely pro HMI".OP_Tocna_4_1_Vyjezd;
      A     "Toèna 4.1 výjezd";
      =     "Události".Tocna_P4_2_Na_Vyjezdu;
END_FUNCTION

FUNCTION "Komunikace" : VOID	// FC 50
VERSION : 0.1
BEGIN
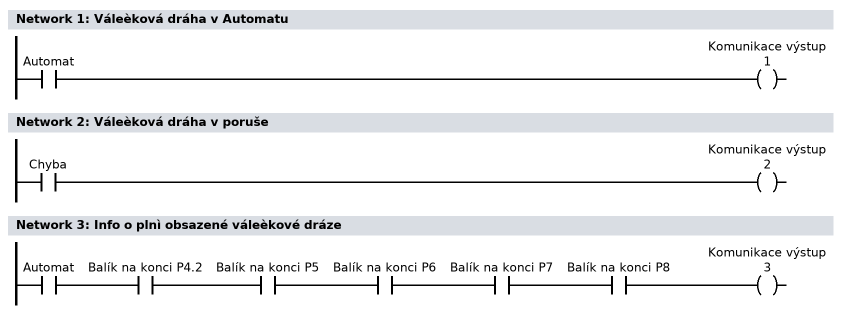
NETWORK
TITLE = Váleèková dráha v Automatu
      A     "Automat";
      =     "Komunikace výstup 1";
NETWORK
TITLE = Váleèková dráha v poruše
      A     "Chyba";
      =     "Komunikace výstup 2";
NETWORK
TITLE = Info o plnì obsazené váleèkové dráze
      A     "Automat";
      A     "Balík na konci P4.2";
      A     "Balík na konci P5";
      A     "Balík na konci P6";
      A     "Balík na konci P7";
      A     "Balík na konci P8";
      =     "Komunikace výstup 3";
END_FUNCTION

DATA_BLOCK "Události"	// DB 100
AUTHOR : Dave
VERSION : 0.1
  STRUCT
   NestandartniOvladani : BOOL ;	//Nestandartni ovladani stroje
   NeniZapnutaSilovka : BOOL ;	//Neni zapnuta silova cast stroje
   Tocna_P2_2_Na_Najezdu : BOOL ;	//Toèna P2.2 je již v pozici nájezdu balíku
   Tocna_P2_2_Na_Vyjezdu : BOOL ;	//Toèna P2.2 je již v pozici výjezdu balíku
   Tocna_P4_2_Na_Najezdu : BOOL ;	//Toèna P4.2 je již v pozici nájezdu balíku
   Tocna_P4_2_Na_Vyjezdu : BOOL ;	//Toèna P4.2 je již v pozici výjezdu balíku
   aaaaa : BOOL ;
   aaaaaa : BOOL ;
   b : BOOL ;
   bb : BOOL ;
   bbb : BOOL ;
   bbbb : BOOL ;
   bbbbb : BOOL ;
   bbbbbb : BOOL ;
   bbbbbbb : BOOL ;
   b7 : BOOL ;
   c : BOOL ;
   c1 : BOOL ;
   c2 : BOOL ;
   c3 : BOOL ;
   c4 : BOOL ;
   c5 : BOOL ;
   c6 : BOOL ;
   c7 : BOOL ;
   d : BOOL ;
   d1 : BOOL ;
   D2 : BOOL ;
   d3 : BOOL ;
   d4 : BOOL ;
   d5 : BOOL ;
   d6 : BOOL ;
   d7 : BOOL ;
   E : DWORD ;
  END_STRUCT ;	
BEGIN
END_DATA_BLOCK

DATA_BLOCK "DB_Chyby"	// DB 101
AUTHOR : Dave
VERSION : 0.1
  STRUCT
   Silovka_Dopravy : BOOL ;	//Nejsou zapnuty silové obvody dopravniku
   Jistice_P1_az_P2_2 : BOOL ;	//Spadený jistiè P1 , P2.1 , P2.2
   Jistice_P3_az_P4_2 : BOOL ;	//Spadený jistiè P3 , P4.1 , P4.2
   Jistice_P7_az_P9 : BOOL ;	//Spadený jistiè P7 , P8 , P9
   Central_Stop_Rozvadec : BOOL ;	//Zmáèknuto Central Stop na rozvadìèi
   Central_Stop_1_Doprava : BOOL ;	//Zmáèknuto Central Stop na dopravnících
   Central_Stop_2_Doprava : BOOL ;	//Zmáèknuto Central Stop na dopravnících
   Dlouhy_Presun_Balicka_P2 : BOOL ;	//Pøíliš dlouhý pøesun balíku z balièky na vstupní dopravník
   Dlouhy_Presun_P2_2_P3 : BOOL ;	//Pøíliš dlouhý pøesun balíku z P2.2 na P3
   Dlouhy_Presun_P3_P4_2 : BOOL ;	//Pøíliš dlouhý pøesun balíku z P3 na P4.2
   Dlouhy_Presun_P4_2_P5 : BOOL ;	//Pøíliš dlouhý pøesun balíku z P4.2 na P5
   Dlouhy_Presun_P5_P6 : BOOL ;	//Pøíliš dlouhý pøesun balíku z P5 na P6
   Dlouhy_Presun_P6_P7 : BOOL ;	//Pøíliš dlouhý pøesun balíku z P6 na P7
   Dlouhy_Presun_P7_P8 : BOOL ;	//Pøíliš dlouhý pøesun balíku z P7 na P8
   Dlouhy_Chod_Tocny_P2_2 : BOOL ;	//Pøíliš dlouhý chod otáèení toèny P2.2
   Dlouhy_Chod_Tocny_P4_2 : BOOL ;	//Pøíliš dlouhý chod otáèení toèny P4.2
   Prilis_dlouhy_balik : BOOL ;	//Pøíliš dlouhý balík
   Plna_Valeckova_draha : BOOL ;	//Valeckova draha je preplnena.
   ccc : BOOL ;
   cccc : BOOL ;
   ccccc : BOOL ;
   cccccc : BOOL ;
   ccccccc : BOOL ;
   cccccccc : BOOL ;
   d : BOOL ;
   dd : BOOL ;
   ddd : BOOL ;
   dddd : BOOL ;
   ddddd : BOOL ;
   dddddd : BOOL ;
   ddddddd : BOOL ;
   dddddddd : BOOL ;
   e : BOOL ;
   ee : BOOL ;
   eee : BOOL ;
   eeee : BOOL ;
   eeeee : BOOL ;
   eeeeee : BOOL ;
   eeeeeee : BOOL ;
   eeeeeeee : BOOL ;
   f : BOOL ;
   ff : BOOL ;
   fff : BOOL ;
   ffff : BOOL ;
   fffff : BOOL ;
   ffffff : BOOL ;
   fffffff : BOOL ;
   ffffffff : BOOL ;
   g : BOOL ;
   gg : BOOL ;
   ggg : BOOL ;
   gggg : BOOL ;
   ggggg : BOOL ;
   gggggg : BOOL ;
   ggggggg : BOOL ;
   gggggggg : BOOL ;
   h : BOOL ;
   hh : BOOL ;
   hhh : BOOL ;
   hhhh : BOOL ;
   hhhhh : BOOL ;
   H5 : BOOL ;
   H6 : BOOL ;
   H7 : BOOL ;
   CH : DWORD ;
   I : DWORD ;
  END_STRUCT ;	
BEGIN
END_DATA_BLOCK

DATA_BLOCK "DB_Ruèni povely pro HMI"	// DB 120
VERSION : 0.1
  STRUCT
   OP_Start_Automatu : BOOL ;	//povel z OP start automatu
   OP_Stop_Automatu : BOOL ;	//povel z OP stop automatu
   OP_Manual : BOOL ;	//povel z OP manualní provoz
   OP_Dopravnik_1_Vpred : BOOL ;	//povel z OP dopravnik vpøed
   OP_Tocna_P2_1_Najezd : BOOL ;	//povel z OP toèna nájezd
   OP_Tocna_P2_1_Vyjezd : BOOL ;	//povel z OP toèna výjezd
   OP_Dopravnik_3_Vpred : BOOL ;	//povel z OP dopravnik vpøed
   OP_Dopravnik_4_Vpred : BOOL ;	//povel z OP dopravnik vpøed
   OP_Tocna_4_1_Najezd : BOOL ;	//povel z OP toèna nájezd
   OP_Tocna_4_1_Vyjezd : BOOL ;	//povel z OP toèna výjezd
   OP_Dopravnik_5_Vpred : BOOL ;	//povel z OP dopravnik vpøed
   OP_Dopravnik_6_Vpred : BOOL ;	//povel z OP dopravnik vpøed
   OP_Dopravnik_7_Vpred : BOOL ;	//povel z OP dopravnik vpøed
   OP_Dopravnik_8_Vpred : BOOL ;	//povel z OP dopravnik vpøed
   bbbbbbb : BOOL ;
   bbbbbbbb : BOOL ;
   c : BOOL ;
   cc : BOOL ;
   ccc : BOOL ;
   cccc : BOOL ;
   ccccc : BOOL ;
   cccccc : BOOL ;
   ccccccc : BOOL ;
   cccccccc : BOOL ;
  END_STRUCT ;	
BEGIN
END_DATA_BLOCK

DATA_BLOCK "DB_Data Hmi"	// DB 140
VERSION : 0.1
  STRUCT
   rez : BOOL ;	//zobrazení chyby stroje
   rez1 : BOOL ;	//zobrazení chyby stroje
   rez2 : BOOL ;	//zobrazení chyby stroje
   rez3 : BOOL ;	//zobrazení chyby stroje
   rez4 : BOOL ;	//zobrazení chyby stroje
   rez5 : BOOL ;	//zobrazení chyby stroje
   rez6 : BOOL ;	//zobrazení chyby stroje
   rez7 : BOOL ;	//zobrazení chyby stroje
   rez8 : BOOL ;	//zobrazení chyby stroje
   rez9 : BOOL ;	//zobrazení chyby stroje
   rez10 : BOOL ;	//zobrazení chyby stroje
   rez12 : BOOL ;	//zobrazení chyby stroje
   rez13 : BOOL ;	//zobrazení chyby stroje
   rezerva1 : BOOL ;
   rezerva2 : BOOL ;
   rezerva3 : BOOL ;
   SystemModeDoprava : INT ;
   SystemStatusRezerva : INT ;
   SystemStatusRezerva_1 : INT ;
  END_STRUCT ;	
BEGIN
END_DATA_BLOCK

ORGANIZATION_BLOCK OB 1
TITLE = "Main Program Sweep (Cycle)"
VERSION : 0.1
VAR_TEMP
  OB1_EV_CLASS : BYTE ;	//Bits 0-3 = 1 (Coming event), Bits 4-7 = 1 (Event class 1)
  OB1_SCAN_1 : BYTE ;	//1 (Cold restart scan 1 of OB 1), 3 (Scan 2-n of OB 1)
  OB1_PRIORITY : BYTE ;	//Priority of OB Execution
  OB1_OB_NUMBR : BYTE ;	//1 (Organization block 1, OB1)
  OB1_RESERVED_1 : BYTE ;	//Reserved for system
  OB1_RESERVED_2 : BYTE ;	//Reserved for system
  OB1_PREV_CYCLE : INT ;	//Cycle time of previous OB1 scan (milliseconds)
  OB1_MIN_CYCLE : INT ;	//Minimum cycle time of OB1 (milliseconds)
  OB1_MAX_CYCLE : INT ;	//Maximum cycle time of OB1 (milliseconds)
  OB1_DATE_TIME : DATE_AND_TIME ;	//Date and time OB1 started
END_VAR
BEGIN
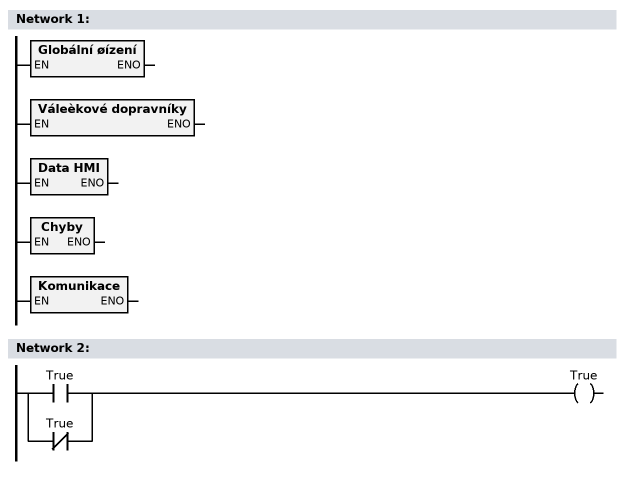
NETWORK
TITLE =
      CALL  "Globální øízení";
      CALL  "Váleèkové dopravníky";
      CALL  "Data HMI";
      CALL  "Chyby";
      CALL  "Komunikace";
NETWORK
TITLE =
      O     "True";
      ON    "True";
      =     "True";
END_ORGANIZATION_BLOCK

ORGANIZATION_BLOCK "CYC_INT5"	// OB 35
TITLE = "Cyclic Interrupt"
VERSION : 0.1
VAR_TEMP
  OB35_EV_CLASS : BYTE ;	//Bits 0-3 = 1 (Coming event), Bits 4-7 = 1 (Event class 1)
  OB35_STRT_INF : BYTE ;	//16#36 (OB 35 has started)
  OB35_PRIORITY : BYTE ;	//Priority of OB Execution
  OB35_OB_NUMBR : BYTE ;	//35 (Organization block 35, OB35)
  OB35_RESERVED_1 : BYTE ;	//Reserved for system
  OB35_RESERVED_2 : BYTE ;	//Reserved for system
  OB35_PHASE_OFFSET : WORD ;	//Phase offset (msec)
  OB35_RESERVED_3 : INT ;	//Reserved for system
  OB35_EXC_FREQ : INT ;	//Frequency of execution (msec)
  OB35_DATE_TIME : DATE_AND_TIME ;	//Date and time OB35 started
END_VAR
BEGIN
// (block stored without names or comments; labels and parameter names are numbered)
END_ORGANIZATION_BLOCK

ORGANIZATION_BLOCK "I/O_FLT1"	// OB 82
TITLE = "I/O Point Fault"
VERSION : 0.1
VAR_TEMP
  OB82_EV_CLASS : BYTE ;	//16#39, Event class 3, Entering event state, Internal fault event
  OB82_FLT_ID : BYTE ;	//16#XX, Fault identifcation code
  OB82_PRIORITY : BYTE ;	//Priority of OB Execution
  OB82_OB_NUMBR : BYTE ;	//82 (Organization block 82, OB82)
  OB82_RESERVED_1 : BYTE ;	//Reserved for system
  OB82_IO_FLAG : BYTE ;	//Input (01010100), Output (01010101)
  OB82_MDL_ADDR : WORD ;	//Base address of module with fault
  OB82_MDL_DEFECT : BOOL ;	//Module defective
  OB82_INT_FAULT : BOOL ;	//Internal fault
  OB82_EXT_FAULT : BOOL ;	//External fault
  OB82_PNT_INFO : BOOL ;	//Point information
  OB82_EXT_VOLTAGE : BOOL ;	//External voltage low
  OB82_FLD_CONNCTR : BOOL ;	//Field wiring connector missing
  OB82_NO_CONFIG : BOOL ;	//Module has no configuration data
  OB82_CONFIG_ERR : BOOL ;	//Module has configuration error
  OB82_MDL_TYPE : BYTE ;	//Type of module
  OB82_SUB_MDL_ERR : BOOL ;	//Sub-Module is missing or has error
  OB82_COMM_FAULT : BOOL ;	//Communication fault
  OB82_MDL_STOP : BOOL ;	//Module is stopped
  OB82_WTCH_DOG_FLT : BOOL ;	//Watch dog timer stopped module
  OB82_INT_PS_FLT : BOOL ;	//Internal power supply fault
  OB82_PRIM_BATT_FLT : BOOL ;	//Primary battery is in fault
  OB82_BCKUP_BATT_FLT : BOOL ;	//Backup battery is in fault
  OB82_RESERVED_2 : BOOL ;	//Reserved for system
  OB82_RACK_FLT : BOOL ;	//Rack fault, only for bus interface module
  OB82_PROC_FLT : BOOL ;	//Processor fault
  OB82_EPROM_FLT : BOOL ;	//EPROM fault
  OB82_RAM_FLT : BOOL ;	//RAM fault
  OB82_ADU_FLT : BOOL ;	//ADU fault
  OB82_FUSE_FLT : BOOL ;	//Fuse fault
  OB82_HW_INTR_FLT : BOOL ;	//Hardware interupt input in fault
  OB82_RESERVED_3 : BOOL ;	//Reserved for system
  OB82_DATE_TIME : DATE_AND_TIME ;	//Date and time OB82 started
END_VAR
BEGIN
// (block stored without names or comments; labels and parameter names are numbered)
END_ORGANIZATION_BLOCK

ORGANIZATION_BLOCK "OBNL_FLT"	// OB 85
TITLE = "Organization Block (OB) Not Loaded Fault"
VERSION : 0.1
VAR_TEMP
  OB85_EV_CLASS : BYTE ;	//16#35 Event class 3
  OB85_FLT_ID : BYTE ;	//16#XX, Fault identification code
  OB85_PRIORITY : BYTE ;	//Priority of OB Execution
  OB85_OB_NUMBR : BYTE ;	//85 (Organization block 85, OB85)
  OB85_RESERVED_1 : BYTE ;	//Reserved for system
  OB85_RESERVED_2 : BYTE ;	//Reserved for system
  OB85_RESERVED_3 : INT ;	//Reserved for system
  OB85_ERR_EV_CLASS : BYTE ;	//Class of event causing error
  OB85_ERR_EV_NUM : BYTE ;	//Number of event causing error
  OB85_OB_PRIOR : BYTE ;	//Priority of OB causing error
  OB85_OB_NUM : BYTE ;	//Number of OB causing error
  OB85_DATE_TIME : DATE_AND_TIME ;	//Date and time OB85 started
END_VAR
BEGIN
// (block stored without names or comments; labels and parameter names are numbered)
END_ORGANIZATION_BLOCK

ORGANIZATION_BLOCK "RACK_FLT"	// OB 86
TITLE = "Loss Of Rack Fault"
VERSION : 0.1
VAR_TEMP
  OB86_EV_CLASS : BYTE ;	//16#38/39 Event class 3
  OB86_FLT_ID : BYTE ;	//16#C1/C4/C5, Fault identifcation code
  OB86_PRIORITY : BYTE ;	//Priority of OB Execution
  OB86_OB_NUMBR : BYTE ;	//86 (Organization block 86, OB86)
  OB86_RESERVED_1 : BYTE ;	//Reserved for system
  OB86_RESERVED_2 : BYTE ;	//Reserved for system
  OB86_MDL_ADDR : WORD ;	//Base address of IM module in rack with fault
  OB86_RACKS_FLTD : ARRAY  [0 .. 31 ] OF BOOL ;	//Racks in fault
  OB86_DATE_TIME : DATE_AND_TIME ;	//Date and time OB86 started
END_VAR
BEGIN
// (block stored without names or comments; labels and parameter names are numbered)
END_ORGANIZATION_BLOCK

ORGANIZATION_BLOCK "Complete Restart"	// OB 100
TITLE = "Complete Restart"
VERSION : 0.1
VAR_TEMP
  OB100_EV_CLASS : BYTE ;	//16#13, Event class 1, Entering event state, Event logged in diagnostic buffer
  OB100_STRTUP : BYTE ;	//16#81/82/83/84 Method of startup
  OB100_PRIORITY : BYTE ;	//Priority of OB Execution
  OB100_OB_NUMBR : BYTE ;	//100 (Organization block 100, OB100)
  OB100_RESERVED_1 : BYTE ;	//Reserved for system
  OB100_RESERVED_2 : BYTE ;	//Reserved for system
  OB100_STOP : WORD ;	//Event that caused CPU to stop (16#4xxx)
  OB100_STRT_INFO : DWORD ;	//Information on how system started
  OB100_DATE_TIME : DATE_AND_TIME ;	//Date and time OB100 started
END_VAR
BEGIN
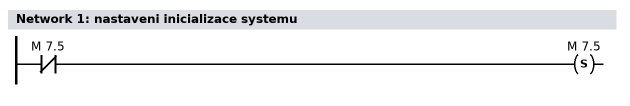
NETWORK
TITLE = nastaveni inicializace systemu
      AN    M 7.5;
      S     M 7.5;
END_ORGANIZATION_BLOCK

ORGANIZATION_BLOCK "Programming Error"	// OB 121
TITLE = "Programming Error"
VERSION : 0.1
VAR_TEMP
  OB121_EV_CLASS : BYTE ;	//16#25, Event class 2, Entering event state, Internal fault event
  OB121_SW_FLT : BYTE ;	//16#XX Software programming fault
  OB121_PRIORITY : BYTE ;	//Priority of OB Execution
  OB121_OB_NUMBR : BYTE ;	//121 (Organization block 121, OB121)
  OB121_BLK_TYPE : BYTE ;	//16#88/8A/8B/8C/8E Type of block fault occured in
  OB121_RESERVED_1 : BYTE ;	//Reserved for system
  OB121_FLT_REG : WORD ;	//16#XX Specific register that caused fault
  OB121_BLK_NUM : WORD ;	//Number of block that programming fault occured in
  OB121_PRG_ADDR : WORD ;	//Address in block where programming fault occured
  OB121_DATE_TIME : DATE_AND_TIME ;	//Date and time OB121 started
END_VAR
BEGIN
// (block stored without names or comments; labels and parameter names are numbered)
END_ORGANIZATION_BLOCK

ORGANIZATION_BLOCK "Module Access Error"	// OB 122
TITLE = "Module Access Error"
VERSION : 0.1
VAR_TEMP
  OB122_EV_CLASS : BYTE ;	//16#29, Event class 2, Entering event state, Internal fault event
  OB122_SW_FLT : BYTE ;	//16#XX Software error code
  OB122_PRIORITY : BYTE ;	//Priority of OB Execution
  OB122_OB_NUMBR : BYTE ;	//122 (Organization block 122, OB122)
  OB122_BLK_TYPE : BYTE ;	//16#88/8C/8E Type of block fault occured in
  OB122_MEM_AREA : BYTE ;	//Memory area where access error occured
  OB122_MEM_ADDR : WORD ;	//Memory address where access error occured
  OB122_BLK_NUM : WORD ;	//Block number in which error occured
  OB122_PRG_ADDR : WORD ;	//Program address where error occured
  OB122_DATE_TIME : DATE_AND_TIME ;	//Date and time OB1 started
END_VAR
BEGIN
// (block stored without names or comments; labels and parameter names are numbered)
END_ORGANIZATION_BLOCK

SYMBOL_TABLE
"Události"	DB 100	DB 100
"DB_Chyby"	DB 101	DB 101
"DB_Ruèni povely pro HMI"	DB 120	DB 120
"DB_Data Hmi"	DB 140	DB 140
"Globální øízení"	FC 10	FC 10
"Váleèkové dopravníky"	FC 20	FC 20
"Data HMI"	FC 30	FC 30
"Chyby"	FC 40	FC 40
"Komunikace"	FC 50	FC 50
"Pohony P1,P2.1 a P2.2 OK"	I 0.0	BOOL	// Pohony dopr.P1 , toèny P2.2 a dopravníku P2.2 jsou OK
"Pohony P3,P4.1 a P4.2 OK"	I 0.1	BOOL	// Pohony dopr.P3 , toèny P4.1 a dopravníku P4.2 jsou OK
"Pohony P7,P8,P9 OK"	I 0.2	BOOL	// Pohony dopr.P7,P8,P9 jsou OK
"Silovka OK"	I 0.3	BOOL	// Silové obvody zapnuty
"Reset"	I 0.4	BOOL	// Reset programu
"Vynut NOT-Aus rozvadìè"	I 0.5	BOOL	// Vypnutý hlavní NOT-AUS na rozvadìèi
"NOT-AUS 1"	I 0.6	BOOL	// Vypnut NOT-AUS 1
"NOT-AUS 2"	I 0.7	BOOL	// Vypnut NOT-AUS 2
"Balík na konci P1"	I 1.0	BOOL	// Balík dojet na konci dopravníku 1
"Balík na konci P2.2"	I 1.1	BOOL	// Balík dojet na konci dopravníku 2.2
"Toèna 2.1 nájezd"	I 1.2	BOOL	// Toèna P2.1 pozice nájezd
"Toèna 2.1 výjezd"	I 1.3	BOOL	// Toèna P2.1 pozice výjezd
"Balík na konci P3"	I 1.4	BOOL	// Balík dojet na konci dopravníku 3
"Balík na konci P4.2"	I 1.5	BOOL	// Balík dojet na konci dopravníku 4.2
"Toèna 4.1 nájezd"	I 1.6	BOOL	// Toèna P4.1 pozice nájezd
"Toèna 4.1 výjezd"	I 1.7	BOOL	// Toèna P4.1 pozice výjezd
"Balík na konci P5"	I 2.0	BOOL	// Balík dojet na konci dopravníku 5
"Balík na konci P6"	I 2.1	BOOL	// Balík dojet na konci dopravníku 6
"Balík na konci P7"	I 2.2	BOOL	// Balík dojet na konci dopravníku 7
"Balík na konci P8"	I 2.3	BOOL	// Balík dojet na konci dopravníku 8
"S024"	I 2.4	BOOL	// stop na D2
"rezerva 1"	I 2.5	BOOL
"rezerva 2"	I 2.6	BOOL
"rezerva 3"	I 2.7	BOOL
"Komunikace vstup 1"	I 3.0	BOOL
"Komunikace vstup2"	I 3.1	BOOL
"Komunikace vstup 3"	I 3.2	BOOL
"Komunikace vstup 4"	I 3.3	BOOL
"rezerva 4"	I 3.4	BOOL
"rezerva 5"	I 3.5	BOOL
"rezerva 6"	I 3.6	BOOL
"rezerva 7"	I 3.7	BOOL
"True"	M 0.3	BOOL
"Automat"	M 1.0	BOOL	// Automatický chod stroje
"Chyba"	M 2.0	BOOL	// vyhlašení chybového stavu stroje
"PM21"	M 2.1	BOOL	// pomocný merkr
"Houkat"	M 4.4	BOOL	// pomocný merkr pro houkaèku
"Toèna P2 Stop nájezd"	M 6.0	BOOL
"Toèna P2 Stop výjezd"	M 6.1	BOOL
"Toèna P4 Stop nájezd"	M 6.2	BOOL
"Toèna P4 Stop výjezd"	M 6.4	BOOL
"M-Toèna 2 nájezd"	M 7.0	BOOL
"M-Toèna 2 výjezd"	M 7.1	BOOL
"M-Toèna 4 výjezd"	M 7.2	BOOL
"M-Toèna 4 nájezd"	M 7.3	BOOL
"Pøesun Balièka-P1"	M 20.0	BOOL	// pomocny merk pøesunu balíku z balièky na toènu
"Pøesun z Toèny na P3"	M 20.1	BOOL	// set a reset pøesunu balíku z toèny na dopravník P3
"Pøesun P3 - Toèna P4."	M 20.2	BOOL	// set a reset pøesunu z dopravníku P3 na toènu P4.1
"Pøesun Toèna P4.1-P5"	M 20.3	BOOL	// set a reset pøesunu z Toèny P4.1 na dopravník P5
"Pøesun P5-P6"	M 20.4	BOOL	// set a reset pøesunu balíku z P5 na P6
"Pøesun P6-P7"	M 20.5	BOOL	// set a reset pøesunu z dopravníku P6 na P7
"Pøesun P7-P8"	M 20.6	BOOL	// set a reset pøesunu z dopravníku P7 na P8
"CYC_INT5"	OB 35	OB 35	// Cyclic Interrupt 5
"I/O_FLT1"	OB 82	OB 82	// I/O Point Fault 1
"OBNL_FLT"	OB 85	OB 85	// OB Not Loaded Fault
"RACK_FLT"	OB 86	OB 86	// Loss of Rack Fault
"Complete Restart"	OB 100	OB 100
"Programming Error"	OB 121	OB 121
"Module Access Error"	OB 122	OB 122
"Dopravník 1 vpøed"	Q 4.0	BOOL	// Start dopravníku 1
"Toèna P2.1 nájezd"	Q 4.1	BOOL	// Toèna P2.1 nájezd
"Toèna P2.1 výjezd"	Q 4.2	BOOL	// Toèna P2.1 výjezd
"Toèna P2.1 brzda"	Q 4.3	BOOL	// Toèna P2.1 bzrda
"Dopravník 2.2 vpøed"	Q 4.4	BOOL	// Start dopravníku 2.2
"Dopravník 3 vpøed"	Q 4.5	BOOL	// Start dopravníku 3
"Toèna P4.1 nájezd"	Q 4.6	BOOL	// Toèna P4.1 nájezd
"Toèna P4.1 výjezd"	Q 4.7	BOOL	// Toèna P4.1 výjezd
"Toèna P4.1 brzda"	Q 5.0	BOOL	// Toèna P4.1 bzrda
"Dopravník P4.2 vpøed"	Q 5.1	BOOL	// Start dopravníku 4.2
"Dopravník 5 vpøed"	Q 5.2	BOOL	// Start dopravníku 5
"Dopravník 6 vpøed"	Q 5.3	BOOL	// Start dopravníku 6
"Dopravník 7 vpøed"	Q 5.4	BOOL	// Start dopravníku 7
"Dopravník 8 vpøed"	Q 5.5	BOOL	// Start dopravníku 8
"rezerva 8"	Q 5.6	BOOL
"rezerva 9"	Q 5.7	BOOL
"Signálka Zapnuto"	Q 6.0	BOOL	// Signálk zapnuto
"rezerva 10"	Q 6.1	BOOL
"rezerva 11"	Q 6.2	BOOL
"rezerva 12"	Q 6.3	BOOL
"Maják zelená"	Q 6.4	BOOL	// Signalizaèní sloupek - zelená
"Maják oranžová"	Q 6.5	BOOL	// Signalizaèní sloupek - oranžová
"Maják èervená"	Q 6.6	BOOL	// Signalizaèní sloupek - èervená
"Houkaèka"	Q 6.7	BOOL	// Signalizaèní sloupek - houkaèka
"Komunikace výstup 1"	Q 7.0	BOOL
"Komunikace výstup 2"	Q 7.1	BOOL
"Komunikace výstup 3"	Q 7.2	BOOL
"Komunikace-Plná linka"	Q 7.3	BOOL
"rezerva 13"	Q 7.4	BOOL
"rezerva 14"	Q 7.5	BOOL
"rezerva 15"	Q 7.6	BOOL
"rezerva 16"	Q 7.7	BOOL
"T-Automat"	T 0	TIMER	// zpoždìné spuštìní automatu
"T-Balík na konci P8"	T 2	TIMER	// Zpoždìný start pøesunu
"T-Pozor"	T 3	TIMER	// upozornìní na spouštìjící se automat
"T-S011"	T 10	TIMER	// balik dojet na konci D2
"T-S015"	T 11	TIMER
"T-Balík na konci"	T 12	TIMER
"T-Možno otoèit toènu"	T 13	TIMER
"T-Možno otoèit toènu P4"	T 14	TIMER
"T-S010"	T 15	TIMER	// balík dojet na konci skluzu
"T-Pøesun Balièka-P2.2"	T 20	TIMER	// èasovaè pro vyhlášení pøíliš dlouhého pøesunu
"T-Pøesun P2.2-P3"	T 21	TIMER	// èasovaè pro vyhlášení pøíliš dlouhého pøesunu
"T-Pøesun P3-P4.2"	T 22	TIMER	// èasovaè pro vyhlášení pøíliš dlouhého pøesunu
"T-Pøesun P4.2-P5"	T 23	TIMER	// èasovaè pro vyhlášení pøíliš dlouhého pøesunu
"T-Pøesun P5-P6"	T 24	TIMER	// èasovaè pro vyhlášení pøíliš dlouhého pøesunu
"T-Pøesun P6-P7"	T 25	TIMER	// èasovaè pro vyhlášení pøíliš dlouhého pøesunu
"T-Pøesun P7-P8"	T 26	TIMER	// èasovaè pro vyhlášení pøíliš dlouhého pøesunu
"T-Otaèení Toèny P2.1"	T 27	TIMER	// èasovaè pro vyhlášení pøíliš dlouhého otáèení toèny
"T-Otáèení toèny P4.1"	T 28	TIMER	// èasovaè pro vyhlášení pøíliš dlouhého otáèení toèny
"T-S014"	T 30	TIMER	// balik dojet na konci dopravniku
"T--S015"	T 31	TIMER	// balík na konci D4
"T-S020"	T 32	TIMER	// balík na konci D5
"T-S021"	T 33	TIMER	// balík na konci D6
"T-S022"	T 34	TIMER	// balík na konci D7
"T--S011"	T 35	TIMER
"T-S024"	T 37	TIMER	// Stop na D2
"T--S014"	T 40	TIMER	// Balík na konci P3
"T--S020"	T 41	TIMER	// Balík na konci P5
"T--S021"	T 42	TIMER	// Balík na konci P6
"T--S022"	T 43	TIMER	// Balík na konci P7
"VAT_1"	VAT 1	
END_SYMBOL_TABLE

FUNCTION "Globální øízení" : VOID	// FC 10
VERSION : 0.1
BEGIN
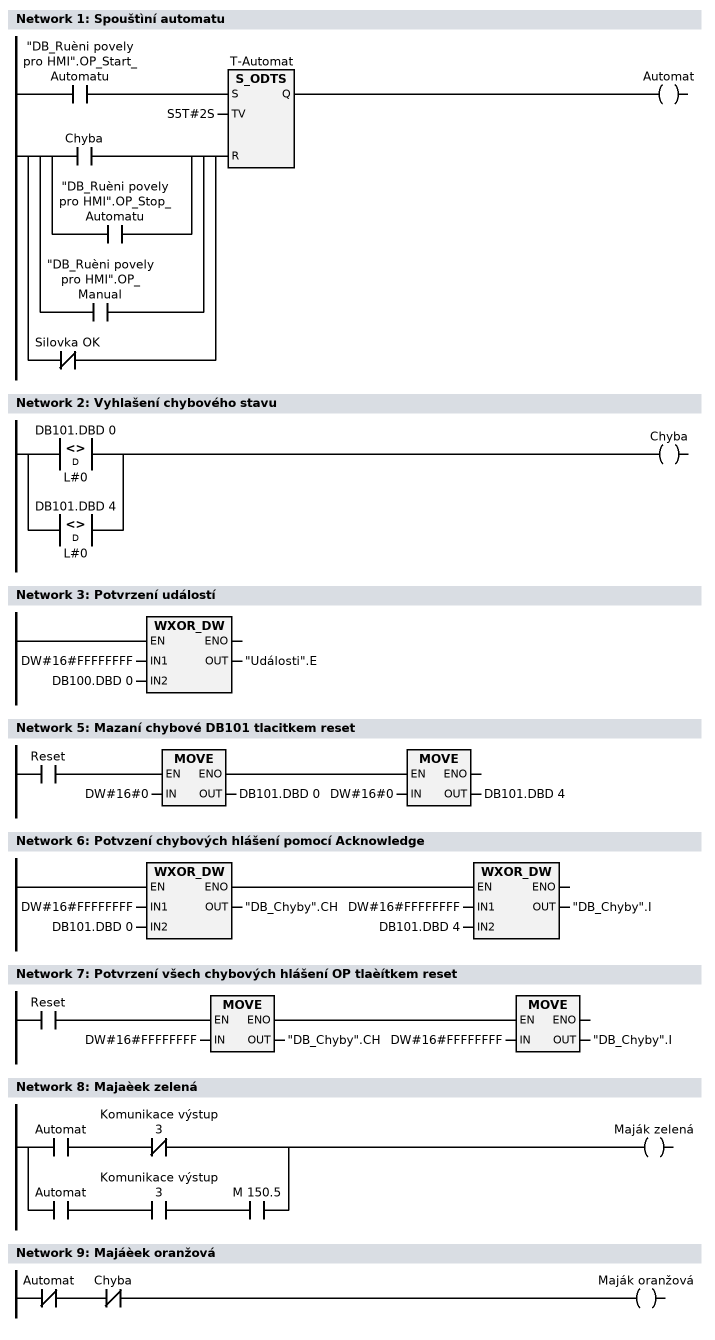
NETWORK
TITLE = Spouštìní automatu 
      A     "DB_Ruèni povely pro HMI".OP_Start_Automatu;
      L     S5T#2S;
      SS    "T-Automat";
      A(;
      O     "Chyba";
      O     "DB_Ruèni povely pro HMI".OP_Stop_Automatu;
      O     "DB_Ruèni povely pro HMI".OP_Manual;
      ON    "Silovka OK";
      );
      R     "T-Automat";
      NOP   0;
      NOP   0;
      A     "T-Automat";
      =     "Automat";
NETWORK
TITLE = Vyhlašení chybového stavu 
      O(;
      L     DB101.DBD 0;
      L     L#0;
      <>D;
      );
      O(;
      L     DB101.DBD 4;
      L     L#0;
      <>D;
      );
      =     "Chyba";
NETWORK
TITLE = Potvrzení událostí
      L     DW#16#FFFFFFFF;
      L     DB100.DBD 0;
      XOD;
      T     "Události".E;
      NOP   0;
NETWORK
TITLE = Akustická signalizace 
      A(;
      O(;
      A     "Chyba";
      FP    "PM21";
      S     "Houkat";
      A     "Reset";
      R     "Houkat";
      A     "Houkat";
      );
      O(;
      A     "DB_Ruèni povely pro HMI".OP_Start_Automatu;
      L     S5T#2S;
      SE    "T-Pozor";
      A(;
      O     "Chyba";
      O     "DB_Ruèni povely pro HMI".OP_Manual;
      O     "DB_Ruèni povely pro HMI".OP_Stop_Automatu;
      O     "Automat";
      );
      R     "T-Pozor";
      NOP   0;
      NOP   0;
      A     "T-Pozor";
      );
      );
      A     M 150.5;
      =     "Houkaèka";
NETWORK
TITLE = Mazaní chybové DB101 tlacitkem reset
      A(;
      A     "Reset";
      JNB   _001;
      L     DW#16#0;
      T     DB101.DBD 0;
      SET;
      SAVE;
      CLR;
_001: A     BR;
      );
      JNB   _002;
      L     DW#16#0;
      T     DB101.DBD 4;
_002: NOP   0;
NETWORK
TITLE = Potvzení chybových hlášení pomocí Acknowledge
      A(;
      L     DW#16#FFFFFFFF;
      L     DB101.DBD 0;
      XOD;
      T     "DB_Chyby".CH;
      SET;
      SAVE;
      CLR;
      A     BR;
      );
      JNB   _003;
      L     DW#16#FFFFFFFF;
      L     DB101.DBD 4;
      XOD;
      T     "DB_Chyby".I;
_003: NOP   0;
NETWORK
TITLE = Potvrzení všech chybových hlášení OP tlaèítkem reset
      A(;
      A     "Reset";
      JNB   _004;
      L     DW#16#FFFFFFFF;
      T     "DB_Chyby".CH;
      SET;
      SAVE;
      CLR;
_004: A     BR;
      );
      JNB   _005;
      L     DW#16#FFFFFFFF;
      T     "DB_Chyby".I;
_005: NOP   0;
NETWORK
TITLE = Majaèek zelená 
      A     "Automat";
      AN    "Komunikace výstup 3";
      O;
      A     "Automat";
      A     "Komunikace výstup 3";
      A     M 150.5;
      =     "Maják zelená";
NETWORK
TITLE = Majáèek oranžová 
      AN    "Automat";
      AN    "Chyba";
      =     "Maják oranžová";
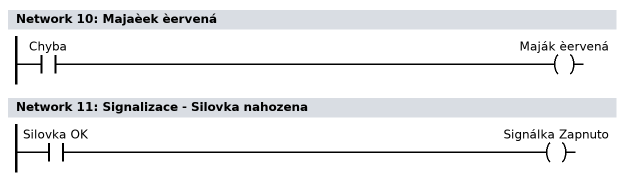
NETWORK
TITLE = Majaèek èervená 
      A     "Chyba";
      =     "Maják èervená";
NETWORK
TITLE = Signalizace - Silovka nahozena
      A     "Silovka OK";
      =     "Signálka Zapnuto";
END_FUNCTION

FUNCTION "Váleèkové dopravníky" : VOID	// FC 20
VERSION : 0.1
BEGIN
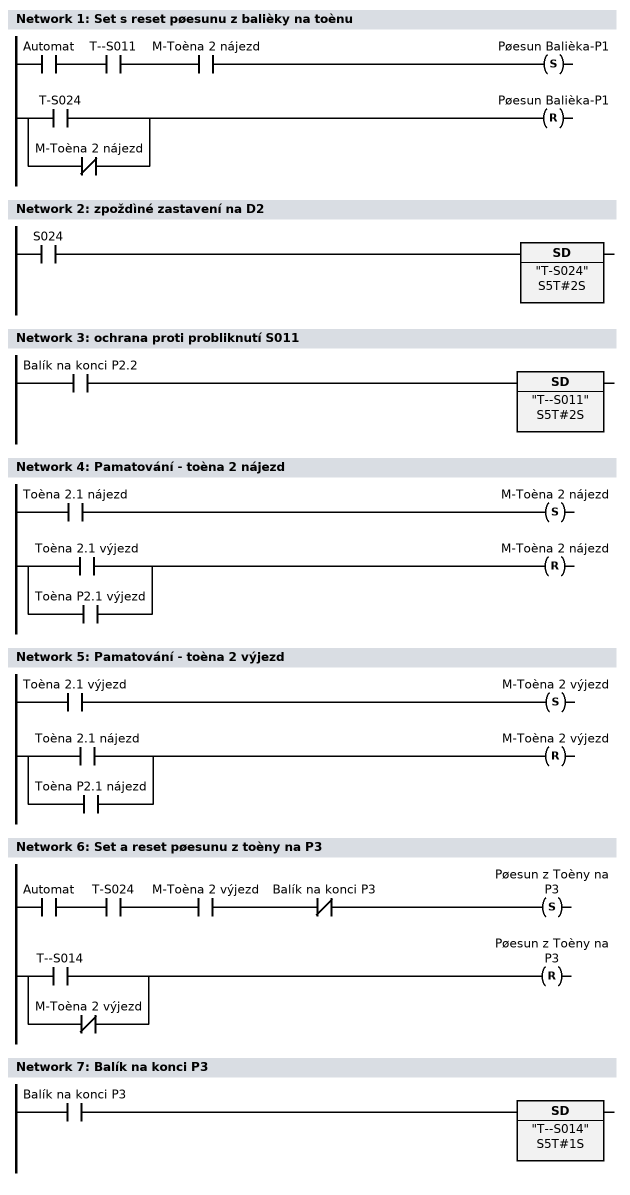
NETWORK
TITLE = Set s reset pøesunu z balièky na toènu
      A     "Automat";
      A     "T--S011";
      A     "M-Toèna 2 nájezd";
      S     "Pøesun Balièka-P1";
      A(;
      O     "T-S024";
      ON    "M-Toèna 2 nájezd";
      );
      R     "Pøesun Balièka-P1";
      NOP   0;
NETWORK
TITLE = zpoždìné zastavení na D2
      A     "S024";
      L     S5T#2S;
      SD    "T-S024";
NETWORK
TITLE = ochrana proti probliknutí S011
      A     "Balík na konci P2.2";
      L     S5T#2S;
      SD    "T--S011";
NETWORK
TITLE = Pamatování - toèna 2 nájezd
      A     "Toèna 2.1 nájezd";
      S     "M-Toèna 2 nájezd";
      A(;
      O     "Toèna 2.1 výjezd";
      O     "Toèna P2.1 výjezd";
      );
      R     "M-Toèna 2 nájezd";
      NOP   0;
NETWORK
TITLE = Pamatování - toèna 2 výjezd
      A     "Toèna 2.1 výjezd";
      S     "M-Toèna 2 výjezd";
      A(;
      O     "Toèna 2.1 nájezd";
      O     "Toèna P2.1 nájezd";
      );
      R     "M-Toèna 2 výjezd";
      NOP   0;
NETWORK
TITLE = Set a reset pøesunu z toèny na P3
      A     "Automat";
      A     "T-S024";
      A     "M-Toèna 2 výjezd";
      AN    "Balík na konci P3";
      S     "Pøesun z Toèny na P3";
      A(;
      O     "T--S014";
      ON    "M-Toèna 2 výjezd";
      );
      R     "Pøesun z Toèny na P3";
      NOP   0;
NETWORK
TITLE = Balík na konci P3
      A     "Balík na konci P3";
      L     S5T#1S;
      SD    "T--S014";
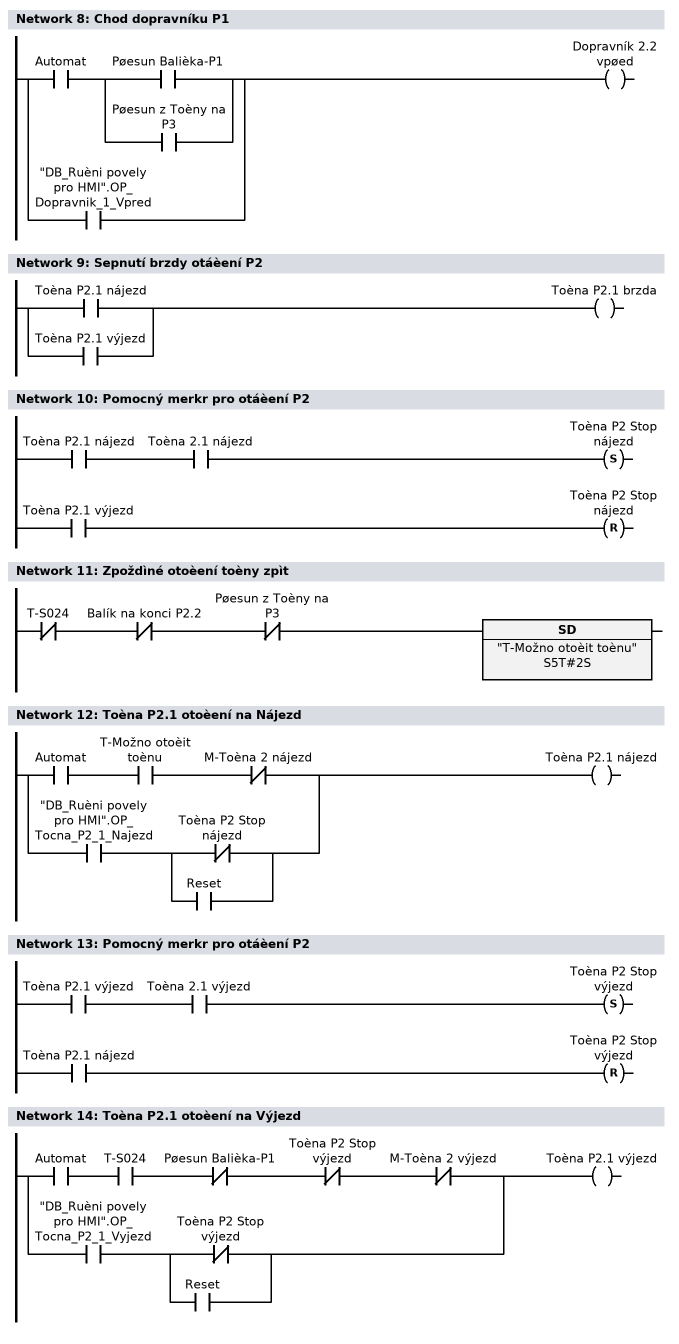
NETWORK
TITLE = Chod dopravníku P1
      A     "Automat";
      A(;
      O     "Pøesun Balièka-P1";
      O     "Pøesun z Toèny na P3";
      );
      O     "DB_Ruèni povely pro HMI".OP_Dopravnik_1_Vpred;
      =     "Dopravník 2.2 vpøed";
NETWORK
TITLE = Sepnutí brzdy otáèení P2
      O     "Toèna P2.1 nájezd";
      O     "Toèna P2.1 výjezd";
      =     "Toèna P2.1 brzda";
NETWORK
TITLE = Pomocný merkr pro otáèení P2
//Kvùli prokmitu toèny 
      A     "Toèna P2.1 nájezd";
      A     "Toèna 2.1 nájezd";
      S     "Toèna P2 Stop nájezd";
      A     "Toèna P2.1 výjezd";
      R     "Toèna P2 Stop nájezd";
      NOP   0;
NETWORK
TITLE = Zpoždìné otoèení toèny zpìt
      AN    "T-S024";
      AN    "Balík na konci P2.2";
      AN    "Pøesun z Toèny na P3";
      L     S5T#2S;
      SD    "T-Možno otoèit toènu";
NETWORK
TITLE = Toèna P2.1 otoèení na Nájezd
      A     "Automat";
      A     "T-Možno otoèit toènu";
      AN    "M-Toèna 2 nájezd";
      O;
      A     "DB_Ruèni povely pro HMI".OP_Tocna_P2_1_Najezd;
      A(;
      ON    "Toèna P2 Stop nájezd";
      O     "Reset";
      );
      =     "Toèna P2.1 nájezd";
NETWORK
TITLE = Pomocný merkr pro otáèení P2
//Kvùli prokmitu toèny 
      A     "Toèna P2.1 výjezd";
      A     "Toèna 2.1 výjezd";
      S     "Toèna P2 Stop výjezd";
      A     "Toèna P2.1 nájezd";
      R     "Toèna P2 Stop výjezd";
      NOP   0;
NETWORK
TITLE = Toèna P2.1 otoèení na Výjezd
      A     "Automat";
      A     "T-S024";
      AN    "Pøesun Balièka-P1";
      AN    "Toèna P2 Stop výjezd";
      AN    "M-Toèna 2 výjezd";
      O;
      A     "DB_Ruèni povely pro HMI".OP_Tocna_P2_1_Vyjezd;
      A(;
      ON    "Toèna P2 Stop výjezd";
      O     "Reset";
      );
      =     "Toèna P2.1 výjezd";
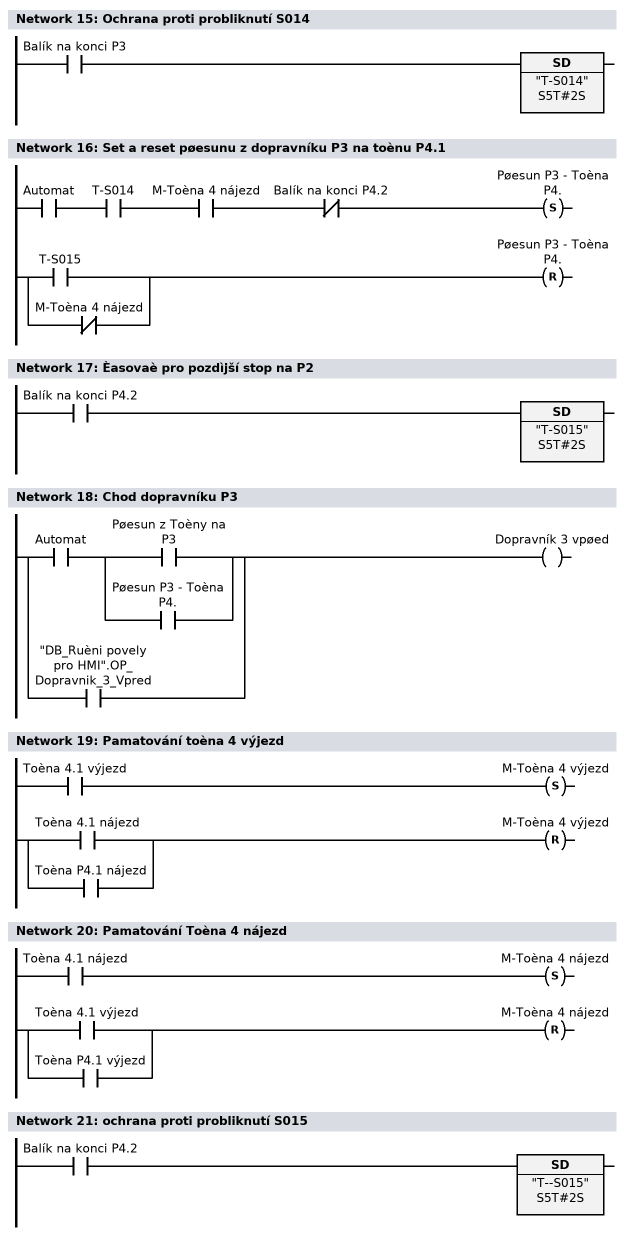
NETWORK
TITLE = Ochrana proti probliknutí S014
      A     "Balík na konci P3";
      L     S5T#2S;
      SD    "T-S014";
NETWORK
TITLE = Set a reset pøesunu z dopravníku P3 na toènu P4.1
      A     "Automat";
      A     "T-S014";
      A     "M-Toèna 4 nájezd";
      AN    "Balík na konci P4.2";
      S     "Pøesun P3 - Toèna P4.";
      A(;
      O     "T-S015";
      ON    "M-Toèna 4 nájezd";
      );
      R     "Pøesun P3 - Toèna P4.";
      NOP   0;
NETWORK
TITLE = Èasovaè pro pozdìjší stop na P2
      A     "Balík na konci P4.2";
      L     S5T#2S;
      SD    "T-S015";
NETWORK
TITLE = Chod dopravníku P3
      A     "Automat";
      A(;
      O     "Pøesun z Toèny na P3";
      O     "Pøesun P3 - Toèna P4.";
      );
      O     "DB_Ruèni povely pro HMI".OP_Dopravnik_3_Vpred;
      =     "Dopravník 3 vpøed";
NETWORK
TITLE = Pamatování toèna 4 výjezd
      A     "Toèna 4.1 výjezd";
      S     "M-Toèna 4 výjezd";
      A(;
      O     "Toèna 4.1 nájezd";
      O     "Toèna P4.1 nájezd";
      );
      R     "M-Toèna 4 výjezd";
      NOP   0;
NETWORK
TITLE = Pamatování Toèna 4 nájezd
      A     "Toèna 4.1 nájezd";
      S     "M-Toèna 4 nájezd";
      A(;
      O     "Toèna 4.1 výjezd";
      O     "Toèna P4.1 výjezd";
      );
      R     "M-Toèna 4 nájezd";
      NOP   0;
NETWORK
TITLE = ochrana proti probliknutí S015
      A     "Balík na konci P4.2";
      L     S5T#2S;
      SD    "T--S015";
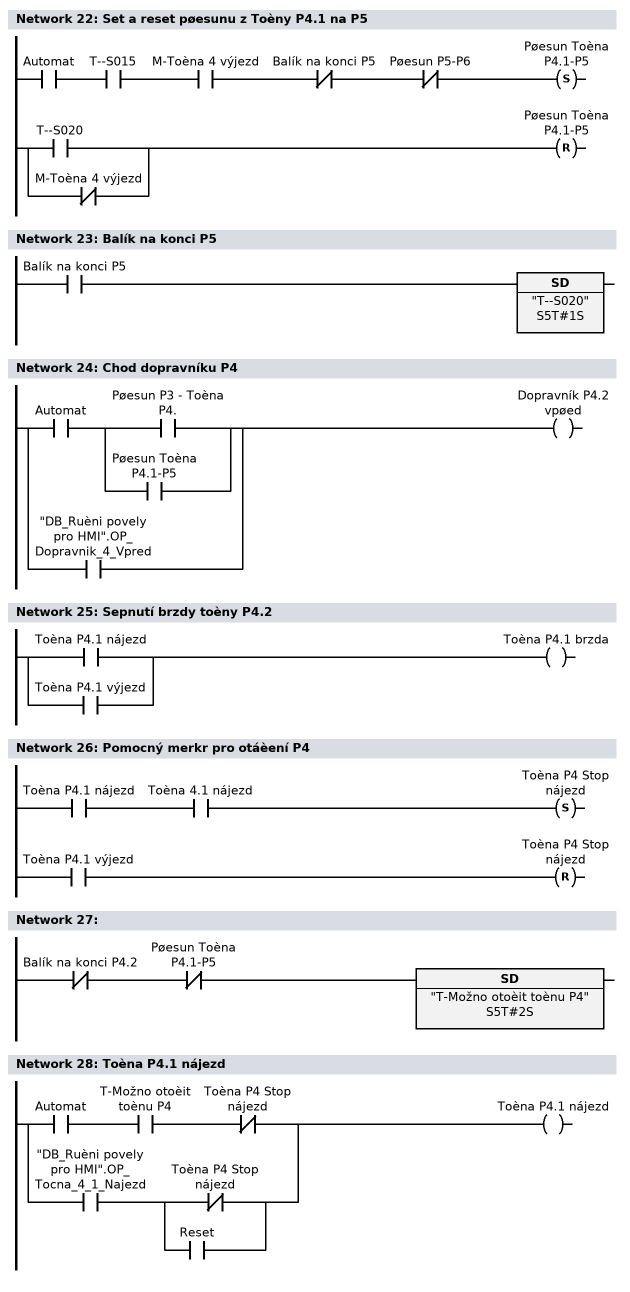
NETWORK
TITLE = Set a reset pøesunu z Toèny P4.1 na P5
      A     "Automat";
      A     "T--S015";
      A     "M-Toèna 4 výjezd";
      AN    "Balík na konci P5";
      AN    "Pøesun P5-P6";
      S     "Pøesun Toèna P4.1-P5";
      A(;
      O     "T--S020";
      ON    "M-Toèna 4 výjezd";
      );
      R     "Pøesun Toèna P4.1-P5";
      NOP   0;
NETWORK
TITLE = Balík na konci P5
      A     "Balík na konci P5";
      L     S5T#1S;
      SD    "T--S020";
NETWORK
TITLE = Chod dopravníku P4
      A     "Automat";
      A(;
      O     "Pøesun P3 - Toèna P4.";
      O     "Pøesun Toèna P4.1-P5";
      );
      O     "DB_Ruèni povely pro HMI".OP_Dopravnik_4_Vpred;
      =     "Dopravník P4.2 vpøed";
NETWORK
TITLE = Sepnutí brzdy toèny P4.2
      O     "Toèna P4.1 nájezd";
      O     "Toèna P4.1 výjezd";
      =     "Toèna P4.1 brzda";
NETWORK
TITLE = Pomocný merkr pro otáèení P4
//
//Kvùli prokmitu toèny 
      A     "Toèna P4.1 nájezd";
      A     "Toèna 4.1 nájezd";
      S     "Toèna P4 Stop nájezd";
      A     "Toèna P4.1 výjezd";
      R     "Toèna P4 Stop nájezd";
      NOP   0;
NETWORK
TITLE =
      AN    "Balík na konci P4.2";
      AN    "Pøesun Toèna P4.1-P5";
      L     S5T#2S;
      SD    "T-Možno otoèit toènu P4";
NETWORK
TITLE = Toèna P4.1 nájezd
      A     "Automat";
      A     "T-Možno otoèit toènu P4";
      AN    "Toèna P4 Stop nájezd";
      O;
      A     "DB_Ruèni povely pro HMI".OP_Tocna_4_1_Najezd;
      A(;
      ON    "Toèna P4 Stop nájezd";
      O     "Reset";
      );
      =     "Toèna P4.1 nájezd";
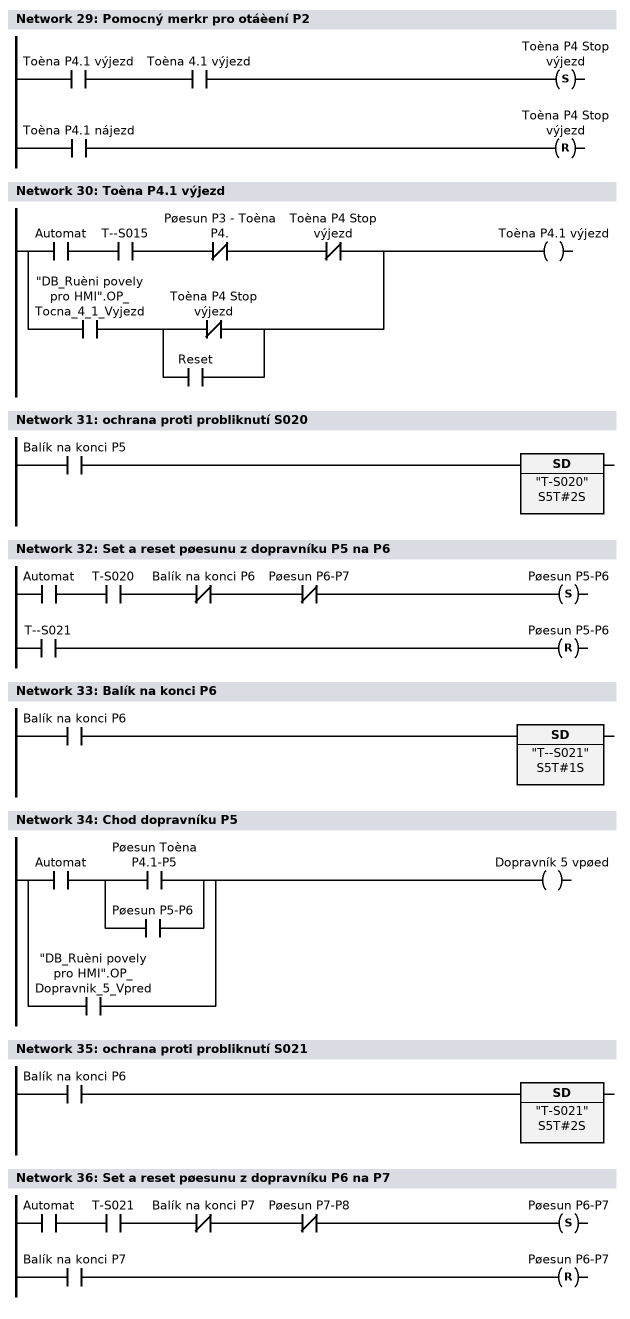
NETWORK
TITLE = Pomocný merkr pro otáèení P2
//Kvùli prokmitu toèny 
      A     "Toèna P4.1 výjezd";
      A     "Toèna 4.1 výjezd";
      S     "Toèna P4 Stop výjezd";
      A     "Toèna P4.1 nájezd";
      R     "Toèna P4 Stop výjezd";
      NOP   0;
NETWORK
TITLE = Toèna P4.1 výjezd
      A     "Automat";
      A     "T--S015";
      AN    "Pøesun P3 - Toèna P4.";
      AN    "Toèna P4 Stop výjezd";
      O;
      A     "DB_Ruèni povely pro HMI".OP_Tocna_4_1_Vyjezd;
      A(;
      ON    "Toèna P4 Stop výjezd";
      O     "Reset";
      );
      =     "Toèna P4.1 výjezd";
NETWORK
TITLE = ochrana proti probliknutí S020
      A     "Balík na konci P5";
      L     S5T#2S;
      SD    "T-S020";
NETWORK
TITLE = Set a reset pøesunu z dopravníku P5 na P6
      A     "Automat";
      A     "T-S020";
      AN    "Balík na konci P6";
      AN    "Pøesun P6-P7";
      S     "Pøesun P5-P6";
      A     "T--S021";
      R     "Pøesun P5-P6";
      NOP   0;
NETWORK
TITLE = Balík na konci P6
      A     "Balík na konci P6";
      L     S5T#1S;
      SD    "T--S021";
NETWORK
TITLE = Chod dopravníku P5
      A     "Automat";
      A(;
      O     "Pøesun Toèna P4.1-P5";
      O     "Pøesun P5-P6";
      );
      O     "DB_Ruèni povely pro HMI".OP_Dopravnik_5_Vpred;
      =     "Dopravník 5 vpøed";
NETWORK
TITLE = ochrana proti probliknutí S021
      A     "Balík na konci P6";
      L     S5T#2S;
      SD    "T-S021";
NETWORK
TITLE = Set a reset pøesunu z dopravníku P6 na P7
      A     "Automat";
      A     "T-S021";
      AN    "Balík na konci P7";
      AN    "Pøesun P7-P8";
      S     "Pøesun P6-P7";
      A     "Balík na konci P7";
      R     "Pøesun P6-P7";
      NOP   0;
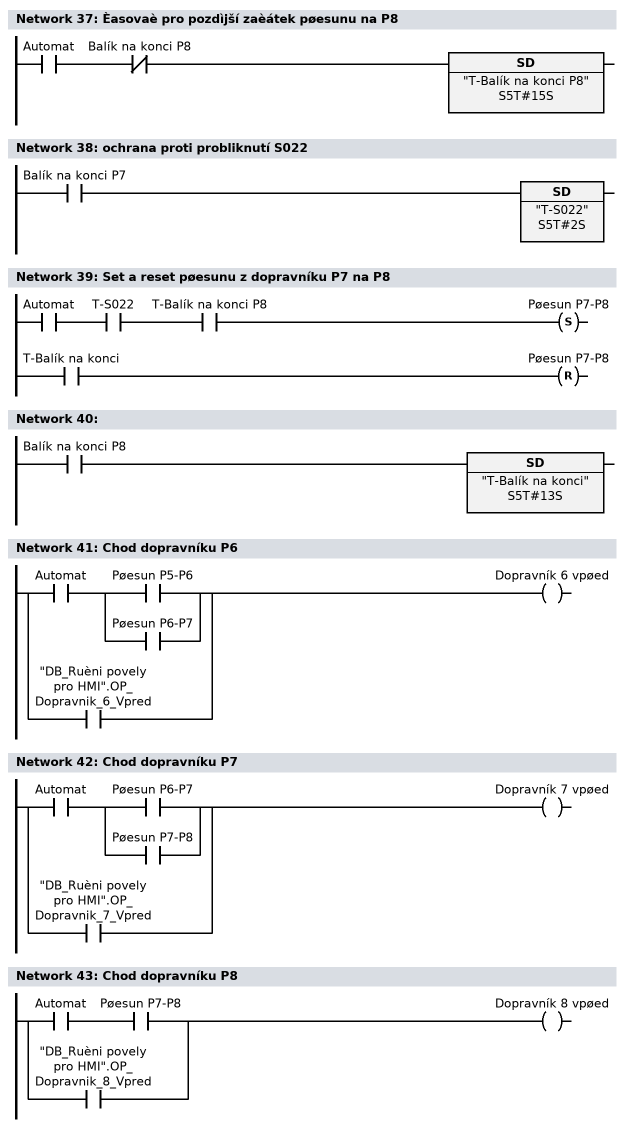
NETWORK
TITLE = Èasovaè pro pozdìjší zaèátek pøesunu na P8
//Je to z dùvodu dání èasu obsluze vozíku na odebrání pøedchozího balíku
      A     "Automat";
      AN    "Balík na konci P8";
      L     S5T#15S;
      SD    "T-Balík na konci P8";
NETWORK
TITLE = ochrana proti probliknutí S022
      A     "Balík na konci P7";
      L     S5T#2S;
      SD    "T-S022";
NETWORK
TITLE = Set a reset pøesunu z dopravníku P7 na P8
      A     "Automat";
      A     "T-S022";
      A     "T-Balík na konci P8";
      S     "Pøesun P7-P8";
      A     "T-Balík na konci";
      R     "Pøesun P7-P8";
      NOP   0;
NETWORK
TITLE =
      A     "Balík na konci P8";
      L     S5T#13S;
      SD    "T-Balík na konci";
NETWORK
TITLE = Chod dopravníku P6
      A     "Automat";
      A(;
      O     "Pøesun P5-P6";
      O     "Pøesun P6-P7";
      );
      O     "DB_Ruèni povely pro HMI".OP_Dopravnik_6_Vpred;
      =     "Dopravník 6 vpøed";
NETWORK
TITLE = Chod dopravníku P7
      A     "Automat";
      A(;
      O     "Pøesun P6-P7";
      O     "Pøesun P7-P8";
      );
      O     "DB_Ruèni povely pro HMI".OP_Dopravnik_7_Vpred;
      =     "Dopravník 7 vpøed";
NETWORK
TITLE = Chod dopravníku P8
      A     "Automat";
      A     "Pøesun P7-P8";
      O     "DB_Ruèni povely pro HMI".OP_Dopravnik_8_Vpred;
      =     "Dopravník 8 vpøed";
END_FUNCTION

FUNCTION "Data HMI" : VOID	// FC 30
VERSION : 0.1
BEGIN
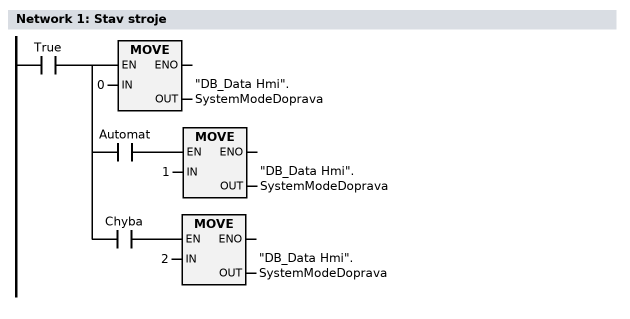
NETWORK
TITLE = Stav stroje 
      A     "True";
      =     L 0.0;
      A     L 0.0;
      JNB   _001;
      L     0;
      T     "DB_Data Hmi".SystemModeDoprava;
_001: NOP   0;
      A     L 0.0;
      A     "Automat";
      JNB   _002;
      L     1;
      T     "DB_Data Hmi".SystemModeDoprava;
_002: NOP   0;
      A     L 0.0;
      A     "Chyba";
      JNB   _003;
      L     2;
      T     "DB_Data Hmi".SystemModeDoprava;
_003: NOP   0;
END_FUNCTION

FUNCTION "Chyby" : VOID	// FC 40
VERSION : 0.1
BEGIN
